SPLINE
SPL {X  -145.877, Y  +737.201, Z    +0.000, E1  +394.468, E3 -286395.030}
SPL {X  -152.550, Y  +719.721, Z    +0.000, E1  +387.728, E3 -286410.519}
SPL {X  -157.145, Y  +701.536, Z    +0.000, E1  +379.368, E3 -286419.974}
SPL {X  -159.035, Y  +688.952, Z    +0.000, E1  +372.676, E3 -286424.015}
SPL {X  -159.873, Y  +677.622, Z    +0.000, E1  +366.008, E3 -286426.087}
SPL {X  -159.990, Y  +671.638, Z    +0.000, E1  +361.925, E3 -286426.713}
SPL {X  -159.990, Y  +668.344, Z    +0.000, E1  +359.382, E3 -286426.906}
SPL {X  -159.990, Y  +664.070, Z    +0.000, E1  +354.975, E3 -286427.234}
SPL {X  -159.990, Y  +656.953, Z    +0.000, E1  +346.040, E3 -286428.300}
SPL {X  -159.990, Y  +644.589, Z    +0.000, E1  +330.989, E3 -286431.712}
SPL {X  -159.990, Y  +605.095, Z    +0.000, E1  +310.486, E3 -286456.803}
SPL {X  -159.990, Y  +546.155, Z    +0.000, E1  +305.539, E3 -286519.561}
SPL {X  -159.990, Y  +539.348, Z    +0.000, E1  +305.531, E3 -286529.865}
SPL {X  -159.990, Y  +530.752, Z    +0.000, E1  +305.518, E3 -286542.872}
SPL {X  -159.990, Y  +522.797, Z    +0.000, E1  +305.537, E3 -286554.956}
SPL {X  -159.990, Y  +515.332, Z    +0.000, E1  +305.526, E3 -286566.244}
SPL {X  -159.990, Y  +508.047, Z    +0.000, E1  +305.531, E3 -286577.261}
SPL {X  -159.990, Y  +499.403, Z    +0.000, E1  +305.488, E3 -286590.300}
SPL {X  -159.990, Y  +479.413, Z    +0.000, E1  +302.719, E3 -286601.446}
SPL {X  -159.990, Y  +454.926, Z    +0.000, E1  +299.433, E3 -286610.552}
SPL {X  -159.990, Y  +449.697, Z    +0.000, E1  +300.191, E3 -286622.015}
SPL {X  -159.990, Y  +444.026, Z    +0.000, E1  +301.072, E3 -286635.273}
SPL {X  -159.990, Y  +437.596, Z    +0.000, E1  +301.764, E3 -286648.015}
SPL {X  -159.990, Y  +432.883, Z    +0.000, E1  +302.386, E3 -286658.411}
SPL {X  -159.990, Y  +429.044, Z    +0.000, E1  +303.109, E3 -286668.302}
SPL {X  -159.990, Y  +425.222, Z    +0.000, E1  +304.101, E3 -286680.199}
SPL {X  -159.990, Y  +418.562, Z    +0.000, E1  +304.950, E3 -286695.356}
SPL {X  -159.990, Y  +410.722, Z    +0.000, E1  +305.100, E3 -286707.817}
SPL {X  -159.990, Y  +402.790, Z    +0.000, E1  +305.070, E3 -286719.592}
SPL {X  -159.990, Y  +391.119, Z    +0.000, E1  +305.052, E3 -286736.970}
SPL {X  -159.988, Y  +381.720, Z    +0.000, E1  +305.103, E3 -286751.077}
SPL {X  -159.786, Y  +374.425, Z    +0.000, E1  +305.121, E3 -286762.125}
SPL {X  -159.015, Y  +364.863, Z    +0.000, E1  +305.220, E3 -286777.142}
SPL {X  -157.966, Y  +357.131, Z    +0.000, E1  +305.441, E3 -286789.832}
SPL {X  -156.775, Y  +350.586, Z    +0.000, E1  +305.627, E3 -286800.806}
SPL {X  -155.397, Y  +344.442, Z    +0.000, E1  +305.886, E3 -286811.422}
SPL {X  -153.976, Y  +339.046, Z    +0.000, E1  +306.128, E3 -286820.914}
SPL {X  -152.417, Y  +333.859, Z    +0.000, E1  +306.416, E3 -286830.240}
SPL {X  -150.681, Y  +328.723, Z    +0.000, E1  +306.710, E3 -286839.616}
SPL {X  -148.661, Y  +323.366, Z    +0.000, E1  +307.100, E3 -286849.625}
SPL {X  -147.089, Y  +319.560, Z    +0.000, E1  +307.396, E3 -286856.840}
SPL {X  -145.161, Y  +315.232, Z    +0.000, E1  +307.745, E3 -286865.121}
SPL {X  -142.534, Y  +309.830, Z    +0.000, E1  +308.237, E3 -286875.626}
SPL {X  -132.342, Y  +292.599, Z    +0.000, E1  +315.826, E3 -286972.914}
ENDSPLINE

SPLINE
SPL {X  -151.238, Y  +330.309, Z    +0.000, E1  +330.693, E3 -287046.071}
SPL {X  -156.949, Y  +351.453, Z    +0.000, E1  +340.161, E3 -287058.231}
SPL {X  -159.024, Y  +364.945, Z    +0.000, E1  +347.297, E3 -287062.649}
SPL {X  -159.758, Y  +373.891, Z    +0.000, E1  +352.513, E3 -287064.538}
SPL {X  -159.985, Y  +381.208, Z    +0.000, E1  +357.184, E3 -287065.421}
SPL {X  -159.990, Y  +385.261, Z    +0.000, E1  +360.259, E3 -287065.691}
SPL {X  -159.990, Y  +388.094, Z    +0.000, E1  +363.012, E3 -287065.883}
SPL {X  -159.990, Y  +390.622, Z    +0.000, E1  +365.876, E3 -287066.122}
SPL {X  -159.990, Y  +394.493, Z    +0.000, E1  +370.512, E3 -287066.645}
SPL {X  -159.990, Y  +401.377, Z    +0.000, E1  +379.398, E3 -287068.099}
SPL {X  -159.990, Y  +411.365, Z    +0.000, E1  +390.630, E3 -287071.307}
SPL {X  -159.990, Y  +450.467, Z    +0.000, E1  +410.183, E3 -287094.956}
SPL {X  -159.990, Y  +509.934, Z    +0.000, E1  +414.923, E3 -287157.575}
SPL {X  -159.990, Y  +516.848, Z    +0.000, E1  +414.930, E3 -287167.863}
SPL {X  -159.990, Y  +524.818, Z    +0.000, E1  +414.933, E3 -287179.735}
SPL {X  -159.990, Y  +532.100, Z    +0.000, E1  +414.924, E3 -287190.588}
SPL {X  -159.990, Y  +539.391, Z    +0.000, E1  +414.933, E3 -287201.440}
SPL {X  -159.990, Y  +546.283, Z    +0.000, E1  +414.924, E3 -287211.712}
SPL {X  -159.990, Y  +553.734, Z    +0.000, E1  +414.938, E3 -287222.799}
SPL {X  -159.990, Y  +564.956, Z    +0.000, E1  +414.973, E3 -287239.470}
SPL {X  -159.990, Y  +577.902, Z    +0.000, E1  +414.969, E3 -287258.760}
SPL {X  -159.990, Y  +588.063, Z    +0.000, E1  +414.931, E3 -287273.951}
SPL {X  -159.990, Y  +595.273, Z    +0.000, E1  +414.928, E3 -287284.674}
SPL {X  -159.990, Y  +602.326, Z    +0.000, E1  +414.932, E3 -287295.174}
SPL {X  -159.990, Y  +609.708, Z    +0.000, E1  +414.930, E3 -287306.181}
SPL {X  -159.990, Y  +618.088, Z    +0.000, E1  +414.948, E3 -287318.610}
SPL {X  -159.990, Y  +625.928, Z    +0.000, E1  +414.931, E3 -287330.306}
SPL {X  -159.990, Y  +632.991, Z    +0.000, E1  +414.938, E3 -287340.809}
SPL {X  -159.990, Y  +639.033, Z    +0.000, E1  +414.931, E3 -287349.817}
SPL {X  -159.990, Y  +646.303, Z    +0.000, E1  +414.946, E3 -287360.604}
SPL {X  -159.990, Y  +656.335, Z    +0.000, E1  +414.969, E3 -287375.507}
SPL {X  -159.990, Y  +664.577, Z    +0.000, E1  +414.924, E3 -287387.884}
SPL {X  -159.989, Y  +672.128, Z    +0.000, E1  +414.946, E3 -287399.101}
SPL {X  -159.792, Y  +679.466, Z    +0.000, E1  +414.893, E3 -287410.259}
SPL {X  -159.330, Y  +686.016, Z    +0.000, E1  +414.837, E3 -287420.490}
SPL {X  -158.190, Y  +695.432, Z    +0.000, E1  +414.658, E3 -287435.686}
SPL {X  -157.027, Y  +702.151, Z    +0.000, E1  +414.415, E3 -287446.968}
SPL {X  -156.112, Y  +706.513, Z    +0.000, E1  +414.265, E3 -287454.402}
SPL {X  -154.917, Y  +711.470, Z    +0.000, E1  +414.052, E3 -287463.030}
SPL {X  -153.561, Y  +716.398, Z    +0.000, E1  +413.816, E3 -287471.751}
SPL {X  -151.715, Y  +722.287, Z    +0.000, E1  +413.503, E3 -287482.367}
SPL {X  -148.967, Y  +729.859, Z    +0.000, E1  +413.026, E3 -287496.359}
SPL {X  -145.862, Y  +737.236, Z    +0.000, E1  +412.427, E3 -287510.414}
SPL {X  -142.777, Y  +743.691, Z    +0.000, E1  +411.831, E3 -287522.957}
SPL {X  -132.301, Y  +761.463, Z    +0.000, E1  +405.510, E3 -287602.242}
ENDSPLINE

SPLINE
SPL {X  -145.877, Y  +737.201, Z    +0.000, E1  +394.468, E3 -287685.353}
SPL {X  -152.550, Y  +719.721, Z    +0.000, E1  +387.728, E3 -287700.842}
SPL {X  -157.145, Y  +701.536, Z    +0.000, E1  +379.368, E3 -287710.296}
SPL {X  -159.035, Y  +688.952, Z    +0.000, E1  +372.676, E3 -287714.337}
SPL {X  -159.756, Y  +680.154, Z    +0.000, E1  +367.520, E3 -287716.064}
SPL {X  -159.986, Y  +672.560, Z    +0.000, E1  +362.636, E3 -287716.962}
SPL {X  -159.990, Y  +668.344, Z    +0.000, E1  +359.382, E3 -287717.228}
SPL {X  -159.990, Y  +664.070, Z    +0.000, E1  +354.975, E3 -287717.556}
SPL {X  -159.990, Y  +656.953, Z    +0.000, E1  +346.040, E3 -287718.623}
SPL {X  -159.990, Y  +644.589, Z    +0.000, E1  +330.989, E3 -287722.034}
SPL {X  -159.990, Y  +605.095, Z    +0.000, E1  +310.486, E3 -287747.125}
SPL {X  -159.990, Y  +546.155, Z    +0.000, E1  +305.539, E3 -287809.884}
SPL {X  -159.990, Y  +539.348, Z    +0.000, E1  +305.531, E3 -287820.188}
SPL {X  -159.990, Y  +530.752, Z    +0.000, E1  +305.518, E3 -287833.195}
SPL {X  -159.990, Y  +522.797, Z    +0.000, E1  +305.537, E3 -287845.278}
SPL {X  -159.990, Y  +515.332, Z    +0.000, E1  +305.526, E3 -287856.567}
SPL {X  -159.990, Y  +508.047, Z    +0.000, E1  +305.531, E3 -287867.584}
SPL {X  -159.990, Y  +499.403, Z    +0.000, E1  +305.488, E3 -287880.623}
SPL {X  -159.990, Y  +479.413, Z    +0.000, E1  +302.719, E3 -287891.768}
SPL {X  -159.990, Y  +454.926, Z    +0.000, E1  +299.433, E3 -287900.875}
SPL {X  -159.990, Y  +449.697, Z    +0.000, E1  +300.191, E3 -287912.337}
SPL {X  -159.990, Y  +445.847, Z    +0.000, E1  +300.905, E3 -287921.960}
SPL {X  -159.990, Y  +439.266, Z    +0.000, E1  +301.568, E3 -287935.044}
SPL {X  -159.990, Y  +432.883, Z    +0.000, E1  +302.386, E3 -287948.734}
SPL {X  -159.990, Y  +429.044, Z    +0.000, E1  +303.109, E3 -287958.624}
SPL {X  -159.990, Y  +425.222, Z    +0.000, E1  +304.101, E3 -287970.521}
SPL {X  -159.990, Y  +420.083, Z    +0.000, E1  +304.918, E3 -287983.097}
SPL {X  -159.990, Y  +412.567, Z    +0.000, E1  +305.072, E3 -287995.321}
SPL {X  -159.990, Y  +402.790, Z    +0.000, E1  +305.070, E3 -288009.915}
SPL {X  -159.990, Y  +391.119, Z    +0.000, E1  +305.052, E3 -288027.293}
SPL {X  -159.988, Y  +381.720, Z    +0.000, E1  +305.103, E3 -288041.400}
SPL {X  -159.786, Y  +374.425, Z    +0.000, E1  +305.121, E3 -288052.448}
SPL {X  -159.015, Y  +364.863, Z    +0.000, E1  +305.220, E3 -288067.464}
SPL {X  -157.966, Y  +357.131, Z    +0.000, E1  +305.441, E3 -288080.155}
SPL {X  -156.775, Y  +350.586, Z    +0.000, E1  +305.627, E3 -288091.129}
SPL {X  -155.027, Y  +342.959, Z    +0.000, E1  +305.926, E3 -288104.302}
SPL {X  -152.882, Y  +335.340, Z    +0.000, E1  +306.305, E3 -288117.844}
SPL {X  -150.681, Y  +328.723, Z    +0.000, E1  +306.710, E3 -288129.939}
SPL {X  -148.661, Y  +323.366, Z    +0.000, E1  +307.100, E3 -288139.948}
SPL {X  -147.089, Y  +319.560, Z    +0.000, E1  +307.396, E3 -288147.163}
SPL {X  -145.161, Y  +315.232, Z    +0.000, E1  +307.745, E3 -288155.443}
SPL {X  -142.534, Y  +309.830, Z    +0.000, E1  +308.237, E3 -288165.948}
SPL {X  -132.342, Y  +292.599, Z    +0.000, E1  +315.826, E3 -288263.237}
ENDSPLINE

SPLINE
SPL {X  -151.238, Y  +330.309, Z    +0.000, E1  +330.693, E3 -288336.393}
SPL {X  -156.949, Y  +351.453, Z    +0.000, E1  +340.161, E3 -288348.554}
SPL {X  -159.024, Y  +364.945, Z    +0.000, E1  +347.297, E3 -288352.972}
SPL {X  -159.878, Y  +376.512, Z    +0.000, E1  +354.071, E3 -288355.223}
SPL {X  -159.990, Y  +383.659, Z    +0.000, E1  +358.950, E3 -288355.918}
SPL {X  -159.990, Y  +387.327, Z    +0.000, E1  +362.137, E3 -288356.151}
SPL {X  -159.990, Y  +390.622, Z    +0.000, E1  +365.876, E3 -288356.444}
SPL {X  -159.990, Y  +394.493, Z    +0.000, E1  +370.512, E3 -288356.967}
SPL {X  -159.990, Y  +401.377, Z    +0.000, E1  +379.398, E3 -288358.422}
SPL {X  -159.990, Y  +411.365, Z    +0.000, E1  +390.630, E3 -288361.630}
SPL {X  -159.990, Y  +450.467, Z    +0.000, E1  +410.183, E3 -288385.279}
SPL {X  -159.990, Y  +509.934, Z    +0.000, E1  +414.923, E3 -288447.898}
SPL {X  -159.990, Y  +516.848, Z    +0.000, E1  +414.930, E3 -288458.186}
SPL {X  -159.990, Y  +524.818, Z    +0.000, E1  +414.933, E3 -288470.058}
SPL {X  -159.990, Y  +532.100, Z    +0.000, E1  +414.924, E3 -288480.911}
SPL {X  -159.990, Y  +539.391, Z    +0.000, E1  +414.933, E3 -288491.763}
SPL {X  -159.990, Y  +546.283, Z    +0.000, E1  +414.924, E3 -288502.034}
SPL {X  -159.990, Y  +553.734, Z    +0.000, E1  +414.938, E3 -288513.121}
SPL {X  -159.990, Y  +564.956, Z    +0.000, E1  +414.973, E3 -288529.792}
SPL {X  -159.990, Y  +577.902, Z    +0.000, E1  +414.969, E3 -288549.082}
SPL {X  -159.990, Y  +588.063, Z    +0.000, E1  +414.931, E3 -288564.273}
SPL {X  -159.990, Y  +595.273, Z    +0.000, E1  +414.928, E3 -288574.997}
SPL {X  -159.990, Y  +602.326, Z    +0.000, E1  +414.932, E3 -288585.497}
SPL {X  -159.990, Y  +609.708, Z    +0.000, E1  +414.930, E3 -288596.504}
SPL {X  -159.990, Y  +618.088, Z    +0.000, E1  +414.948, E3 -288608.933}
SPL {X  -159.990, Y  +625.928, Z    +0.000, E1  +414.931, E3 -288620.629}
SPL {X  -159.990, Y  +635.803, Z    +0.000, E1  +414.980, E3 -288635.257}
SPL {X  -159.990, Y  +646.303, Z    +0.000, E1  +414.946, E3 -288650.927}
SPL {X  -159.990, Y  +653.312, Z    +0.000, E1  +414.932, E3 -288661.379}
SPL {X  -159.990, Y  +658.943, Z    +0.000, E1  +414.931, E3 -288669.777}
SPL {X  -159.990, Y  +667.151, Z    +0.000, E1  +414.954, E3 -288681.995}
SPL {X  -159.885, Y  +677.285, Z    +0.000, E1  +414.936, E3 -288697.191}
SPL {X  -159.482, Y  +684.244, Z    +0.000, E1  +414.840, E3 -288708.043}
SPL {X  -158.805, Y  +690.934, Z    +0.000, E1  +414.742, E3 -288718.692}
SPL {X  -157.890, Y  +697.337, Z    +0.000, E1  +414.571, E3 -288729.214}
SPL {X  -156.492, Y  +704.774, Z    +0.000, E1  +414.365, E3 -288741.692}
SPL {X  -154.917, Y  +711.470, Z    +0.000, E1  +414.052, E3 -288753.352}
SPL {X  -153.561, Y  +716.398, Z    +0.000, E1  +413.816, E3 -288762.074}
SPL {X  -151.715, Y  +722.287, Z    +0.000, E1  +413.503, E3 -288772.690}
SPL {X  -148.967, Y  +729.859, Z    +0.000, E1  +413.026, E3 -288786.682}
SPL {X  -145.862, Y  +737.236, Z    +0.000, E1  +412.427, E3 -288800.736}
SPL {X  -142.777, Y  +743.691, Z    +0.000, E1  +411.831, E3 -288813.279}
SPL {X  -132.301, Y  +761.463, Z    +0.000, E1  +405.510, E3 -288892.564}
ENDSPLINE

SPLINE
SPL {X  -145.877, Y  +737.201, Z    +0.000, E1  +394.468, E3 -288975.675}
SPL {X  -152.550, Y  +719.721, Z    +0.000, E1  +387.728, E3 -288991.164}
SPL {X  -157.145, Y  +701.536, Z    +0.000, E1  +379.368, E3 -289000.619}
SPL {X  -159.035, Y  +688.952, Z    +0.000, E1  +372.676, E3 -289004.660}
SPL {X  -159.756, Y  +680.154, Z    +0.000, E1  +367.520, E3 -289006.386}
SPL {X  -159.986, Y  +672.560, Z    +0.000, E1  +362.636, E3 -289007.284}
SPL {X  -159.990, Y  +668.344, Z    +0.000, E1  +359.382, E3 -289007.551}
SPL {X  -159.990, Y  +664.070, Z    +0.000, E1  +354.975, E3 -289007.879}
SPL {X  -159.990, Y  +656.953, Z    +0.000, E1  +346.040, E3 -289008.946}
SPL {X  -159.990, Y  +644.589, Z    +0.000, E1  +330.989, E3 -289012.357}
SPL {X  -159.990, Y  +605.095, Z    +0.000, E1  +310.486, E3 -289037.448}
SPL {X  -159.990, Y  +546.155, Z    +0.000, E1  +305.539, E3 -289100.206}
SPL {X  -159.990, Y  +539.348, Z    +0.000, E1  +305.531, E3 -289110.510}
SPL {X  -159.990, Y  +530.752, Z    +0.000, E1  +305.518, E3 -289123.518}
SPL {X  -159.990, Y  +522.797, Z    +0.000, E1  +305.537, E3 -289135.601}
SPL {X  -159.990, Y  +515.332, Z    +0.000, E1  +305.526, E3 -289146.890}
SPL {X  -159.990, Y  +508.047, Z    +0.000, E1  +305.531, E3 -289157.906}
SPL {X  -159.990, Y  +501.296, Z    +0.000, E1  +305.518, E3 -289168.128}
SPL {X  -159.990, Y  +487.558, Z    +0.000, E1  +304.151, E3 -289179.758}
SPL {X  -159.990, Y  +454.926, Z    +0.000, E1  +299.433, E3 -289191.197}
SPL {X  -159.990, Y  +449.697, Z    +0.000, E1  +300.191, E3 -289202.660}
SPL {X  -159.990, Y  +445.847, Z    +0.000, E1  +300.905, E3 -289212.283}
SPL {X  -159.990, Y  +439.266, Z    +0.000, E1  +301.568, E3 -289225.366}
SPL {X  -159.990, Y  +432.883, Z    +0.000, E1  +302.386, E3 -289239.057}
SPL {X  -159.990, Y  +429.044, Z    +0.000, E1  +303.109, E3 -289248.947}
SPL {X  -159.990, Y  +425.222, Z    +0.000, E1  +304.101, E3 -289260.844}
SPL {X  -159.990, Y  +418.562, Z    +0.000, E1  +304.950, E3 -289276.002}
SPL {X  -159.990, Y  +407.911, Z    +0.000, E1  +305.062, E3 -289292.593}
SPL {X  -159.990, Y  +400.284, Z    +0.000, E1  +305.103, E3 -289304.027}
SPL {X  -159.990, Y  +391.119, Z    +0.000, E1  +305.052, E3 -289317.615}
SPL {X  -159.988, Y  +381.720, Z    +0.000, E1  +305.103, E3 -289331.722}
SPL {X  -159.786, Y  +374.425, Z    +0.000, E1  +305.121, E3 -289342.771}
SPL {X  -159.015, Y  +364.863, Z    +0.000, E1  +305.220, E3 -289357.787}
SPL {X  -157.966, Y  +357.131, Z    +0.000, E1  +305.441, E3 -289370.477}
SPL {X  -156.775, Y  +350.586, Z    +0.000, E1  +305.627, E3 -289381.451}
SPL {X  -155.027, Y  +342.959, Z    +0.000, E1  +305.926, E3 -289394.624}
SPL {X  -152.882, Y  +335.340, Z    +0.000, E1  +306.305, E3 -289408.167}
SPL {X  -150.681, Y  +328.723, Z    +0.000, E1  +306.710, E3 -289420.261}
SPL {X  -148.661, Y  +323.366, Z    +0.000, E1  +307.100, E3 -289430.270}
SPL {X  -147.089, Y  +319.560, Z    +0.000, E1  +307.396, E3 -289437.485}
SPL {X  -145.161, Y  +315.232, Z    +0.000, E1  +307.745, E3 -289445.766}
SPL {X  -142.534, Y  +309.830, Z    +0.000, E1  +308.237, E3 -289456.271}
SPL {X  -132.342, Y  +292.599, Z    +0.000, E1  +315.826, E3 -289553.559}
ENDSPLINE

SPLINE
SPL {X  -151.238, Y  +330.309, Z    +0.000, E1  +330.693, E3 -289626.716}
SPL {X  -156.949, Y  +351.453, Z    +0.000, E1  +340.161, E3 -289638.877}
SPL {X  -159.024, Y  +364.945, Z    +0.000, E1  +347.297, E3 -289643.294}
SPL {X  -159.758, Y  +373.891, Z    +0.000, E1  +352.513, E3 -289645.183}
SPL {X  -159.985, Y  +381.208, Z    +0.000, E1  +357.184, E3 -289646.066}
SPL {X  -159.990, Y  +384.493, Z    +0.000, E1  +359.676, E3 -289646.291}
SPL {X  -159.990, Y  +387.327, Z    +0.000, E1  +362.137, E3 -289646.473}
SPL {X  -159.990, Y  +392.053, Z    +0.000, E1  +367.477, E3 -289646.938}
SPL {X  -159.990, Y  +396.158, Z    +0.000, E1  +372.775, E3 -289647.564}
SPL {X  -159.990, Y  +401.377, Z    +0.000, E1  +379.398, E3 -289648.744}
SPL {X  -159.990, Y  +411.365, Z    +0.000, E1  +390.630, E3 -289651.953}
SPL {X  -159.990, Y  +450.467, Z    +0.000, E1  +410.183, E3 -289675.602}
SPL {X  -159.990, Y  +509.934, Z    +0.000, E1  +414.923, E3 -289738.220}
SPL {X  -159.990, Y  +516.848, Z    +0.000, E1  +414.930, E3 -289748.508}
SPL {X  -159.990, Y  +524.818, Z    +0.000, E1  +414.933, E3 -289760.380}
SPL {X  -159.990, Y  +532.100, Z    +0.000, E1  +414.924, E3 -289771.233}
SPL {X  -159.990, Y  +539.391, Z    +0.000, E1  +414.933, E3 -289782.085}
SPL {X  -159.990, Y  +546.283, Z    +0.000, E1  +414.924, E3 -289792.357}
SPL {X  -159.990, Y  +553.734, Z    +0.000, E1  +414.938, E3 -289803.444}
SPL {X  -159.990, Y  +564.956, Z    +0.000, E1  +414.973, E3 -289820.115}
SPL {X  -159.990, Y  +577.902, Z    +0.000, E1  +414.969, E3 -289839.405}
SPL {X  -159.990, Y  +588.063, Z    +0.000, E1  +414.931, E3 -289854.596}
SPL {X  -159.990, Y  +595.273, Z    +0.000, E1  +414.928, E3 -289865.319}
SPL {X  -159.990, Y  +602.326, Z    +0.000, E1  +414.932, E3 -289875.820}
SPL {X  -159.990, Y  +609.708, Z    +0.000, E1  +414.930, E3 -289886.826}
SPL {X  -159.990, Y  +618.088, Z    +0.000, E1  +414.948, E3 -289899.255}
SPL {X  -159.990, Y  +625.928, Z    +0.000, E1  +414.931, E3 -289910.951}
SPL {X  -159.990, Y  +635.803, Z    +0.000, E1  +414.980, E3 -289925.579}
SPL {X  -159.990, Y  +646.303, Z    +0.000, E1  +414.946, E3 -289941.250}
SPL {X  -159.990, Y  +656.335, Z    +0.000, E1  +414.969, E3 -289956.152}
SPL {X  -159.990, Y  +664.577, Z    +0.000, E1  +414.924, E3 -289968.529}
SPL {X  -159.989, Y  +672.128, Z    +0.000, E1  +414.946, E3 -289979.746}
SPL {X  -159.636, Y  +682.136, Z    +0.000, E1  +414.901, E3 -289995.004}
SPL {X  -158.805, Y  +690.934, Z    +0.000, E1  +414.742, E3 -290009.015}
SPL {X  -157.890, Y  +697.337, Z    +0.000, E1  +414.571, E3 -290019.536}
SPL {X  -156.492, Y  +704.774, Z    +0.000, E1  +414.365, E3 -290032.015}
SPL {X  -154.917, Y  +711.470, Z    +0.000, E1  +414.052, E3 -290043.675}
SPL {X  -153.204, Y  +717.603, Z    +0.000, E1  +413.775, E3 -290054.521}
SPL {X  -151.355, Y  +723.351, Z    +0.000, E1  +413.415, E3 -290064.992}
SPL {X  -148.967, Y  +729.859, Z    +0.000, E1  +413.026, E3 -290077.004}
SPL {X  -145.862, Y  +737.236, Z    +0.000, E1  +412.427, E3 -290091.059}
SPL {X  -142.777, Y  +743.691, Z    +0.000, E1  +411.831, E3 -290103.602}
SPL {X  -132.301, Y  +761.463, Z    +0.000, E1  +405.510, E3 -290182.887}
ENDSPLINE

SPLINE
SPL {X  -145.877, Y  +737.201, Z    +0.000, E1  +394.468, E3 -290265.998}
SPL {X  -152.550, Y  +719.721, Z    +0.000, E1  +387.728, E3 -290281.487}
SPL {X  -157.145, Y  +701.536, Z    +0.000, E1  +379.368, E3 -290290.942}
SPL {X  -159.035, Y  +688.952, Z    +0.000, E1  +372.676, E3 -290294.983}
SPL {X  -159.756, Y  +680.154, Z    +0.000, E1  +367.520, E3 -290296.709}
SPL {X  -159.986, Y  +672.560, Z    +0.000, E1  +362.636, E3 -290297.607}
SPL {X  -159.990, Y  +669.364, Z    +0.000, E1  +360.170, E3 -290297.815}
SPL {X  -159.990, Y  +667.647, Z    +0.000, E1  +358.660, E3 -290297.913}
SPL {X  -159.990, Y  +664.070, Z    +0.000, E1  +354.975, E3 -290298.202}
SPL {X  -159.990, Y  +656.953, Z    +0.000, E1  +346.040, E3 -290299.268}
SPL {X  -159.990, Y  +644.589, Z    +0.000, E1  +330.989, E3 -290302.680}
SPL {X  -159.990, Y  +605.095, Z    +0.000, E1  +310.486, E3 -290327.771}
SPL {X  -159.990, Y  +546.155, Z    +0.000, E1  +305.539, E3 -290390.529}
SPL {X  -159.990, Y  +539.348, Z    +0.000, E1  +305.531, E3 -290400.833}
SPL {X  -159.990, Y  +530.752, Z    +0.000, E1  +305.518, E3 -290413.840}
SPL {X  -159.990, Y  +522.797, Z    +0.000, E1  +305.537, E3 -290425.923}
SPL {X  -159.990, Y  +515.332, Z    +0.000, E1  +305.526, E3 -290437.212}
SPL {X  -159.990, Y  +508.047, Z    +0.000, E1  +305.531, E3 -290448.229}
SPL {X  -159.990, Y  +499.403, Z    +0.000, E1  +305.488, E3 -290461.268}
SPL {X  -159.990, Y  +479.413, Z    +0.000, E1  +302.719, E3 -290472.413}
SPL {X  -159.990, Y  +454.926, Z    +0.000, E1  +299.433, E3 -290481.520}
SPL {X  -159.990, Y  +449.697, Z    +0.000, E1  +300.191, E3 -290492.982}
SPL {X  -159.990, Y  +445.847, Z    +0.000, E1  +300.905, E3 -290502.605}
SPL {X  -159.990, Y  +439.266, Z    +0.000, E1  +301.568, E3 -290515.689}
SPL {X  -159.990, Y  +432.883, Z    +0.000, E1  +302.386, E3 -290529.379}
SPL {X  -159.990, Y  +429.044, Z    +0.000, E1  +303.109, E3 -290539.269}
SPL {X  -159.990, Y  +425.222, Z    +0.000, E1  +304.101, E3 -290551.166}
SPL {X  -159.990, Y  +420.083, Z    +0.000, E1  +304.918, E3 -290563.742}
SPL {X  -159.990, Y  +412.567, Z    +0.000, E1  +305.072, E3 -290575.966}
SPL {X  -159.990, Y  +402.790, Z    +0.000, E1  +305.070, E3 -290590.560}
SPL {X  -159.990, Y  +391.119, Z    +0.000, E1  +305.052, E3 -290607.938}
SPL {X  -159.988, Y  +381.720, Z    +0.000, E1  +305.103, E3 -290622.045}
SPL {X  -159.786, Y  +374.425, Z    +0.000, E1  +305.121, E3 -290633.093}
SPL {X  -159.015, Y  +364.863, Z    +0.000, E1  +305.220, E3 -290648.109}
SPL {X  -157.966, Y  +357.131, Z    +0.000, E1  +305.441, E3 -290660.800}
SPL {X  -156.775, Y  +350.586, Z    +0.000, E1  +305.627, E3 -290671.774}
SPL {X  -155.027, Y  +342.959, Z    +0.000, E1  +305.926, E3 -290684.947}
SPL {X  -152.882, Y  +335.340, Z    +0.000, E1  +306.305, E3 -290698.489}
SPL {X  -150.681, Y  +328.723, Z    +0.000, E1  +306.710, E3 -290710.584}
SPL {X  -148.661, Y  +323.366, Z    +0.000, E1  +307.100, E3 -290720.593}
SPL {X  -147.089, Y  +319.560, Z    +0.000, E1  +307.396, E3 -290727.808}
SPL {X  -145.161, Y  +315.232, Z    +0.000, E1  +307.745, E3 -290736.088}
SPL {X  -142.534, Y  +309.830, Z    +0.000, E1  +308.237, E3 -290746.594}
SPL {X  -132.342, Y  +292.599, Z    +0.000, E1  +315.826, E3 -290843.882}
ENDSPLINE

SPLINE
SPL {X  -151.238, Y  +330.309, Z    +0.000, E1  +330.693, E3 -290917.038}
SPL {X  -156.949, Y  +351.453, Z    +0.000, E1  +340.161, E3 -290929.199}
SPL {X  -159.024, Y  +364.945, Z    +0.000, E1  +347.297, E3 -290933.617}
SPL {X  -159.878, Y  +376.512, Z    +0.000, E1  +354.071, E3 -290935.869}
SPL {X  -159.990, Y  +383.659, Z    +0.000, E1  +358.950, E3 -290936.563}
SPL {X  -159.990, Y  +387.327, Z    +0.000, E1  +362.137, E3 -290936.796}
SPL {X  -159.990, Y  +390.622, Z    +0.000, E1  +365.876, E3 -290937.089}
SPL {X  -159.990, Y  +394.493, Z    +0.000, E1  +370.512, E3 -290937.612}
SPL {X  -159.990, Y  +401.377, Z    +0.000, E1  +379.398, E3 -290939.067}
SPL {X  -159.990, Y  +411.365, Z    +0.000, E1  +390.630, E3 -290942.275}
SPL {X  -159.990, Y  +450.467, Z    +0.000, E1  +410.183, E3 -290965.924}
SPL {X  -159.990, Y  +509.934, Z    +0.000, E1  +414.923, E3 -291028.543}
SPL {X  -159.990, Y  +516.848, Z    +0.000, E1  +414.930, E3 -291038.831}
SPL {X  -159.990, Y  +524.818, Z    +0.000, E1  +414.933, E3 -291050.703}
SPL {X  -159.990, Y  +532.100, Z    +0.000, E1  +414.924, E3 -291061.556}
SPL {X  -159.990, Y  +539.391, Z    +0.000, E1  +414.933, E3 -291072.408}
SPL {X  -159.990, Y  +546.283, Z    +0.000, E1  +414.924, E3 -291082.680}
SPL {X  -159.990, Y  +553.734, Z    +0.000, E1  +414.938, E3 -291093.766}
SPL {X  -159.990, Y  +560.657, Z    +0.000, E1  +414.914, E3 -291104.127}
SPL {X  -159.990, Y  +567.311, Z    +0.000, E1  +414.931, E3 -291114.012}
SPL {X  -159.990, Y  +577.902, Z    +0.000, E1  +414.969, E3 -291129.727}
SPL {X  -159.990, Y  +588.063, Z    +0.000, E1  +414.931, E3 -291144.918}
SPL {X  -159.990, Y  +595.273, Z    +0.000, E1  +414.928, E3 -291155.642}
SPL {X  -159.990, Y  +602.326, Z    +0.000, E1  +414.932, E3 -291166.142}
SPL {X  -159.990, Y  +609.708, Z    +0.000, E1  +414.930, E3 -291177.149}
SPL {X  -159.990, Y  +616.306, Z    +0.000, E1  +414.927, E3 -291186.962}
SPL {X  -159.990, Y  +624.320, Z    +0.000, E1  +414.952, E3 -291198.845}
SPL {X  -159.990, Y  +632.991, Z    +0.000, E1  +414.938, E3 -291211.777}
SPL {X  -159.990, Y  +639.033, Z    +0.000, E1  +414.931, E3 -291220.784}
SPL {X  -159.990, Y  +646.303, Z    +0.000, E1  +414.946, E3 -291231.572}
SPL {X  -159.990, Y  +656.335, Z    +0.000, E1  +414.969, E3 -291246.474}
SPL {X  -159.990, Y  +664.577, Z    +0.000, E1  +414.924, E3 -291258.852}
SPL {X  -159.989, Y  +672.128, Z    +0.000, E1  +414.946, E3 -291270.068}
SPL {X  -159.792, Y  +679.466, Z    +0.000, E1  +414.893, E3 -291281.226}
SPL {X  -159.330, Y  +686.016, Z    +0.000, E1  +414.837, E3 -291291.457}
SPL {X  -158.190, Y  +695.432, Z    +0.000, E1  +414.658, E3 -291306.654}
SPL {X  -157.027, Y  +702.151, Z    +0.000, E1  +414.415, E3 -291317.936}
SPL {X  -156.112, Y  +706.513, Z    +0.000, E1  +414.265, E3 -291325.370}
SPL {X  -154.917, Y  +711.470, Z    +0.000, E1  +414.052, E3 -291333.997}
SPL {X  -153.561, Y  +716.398, Z    +0.000, E1  +413.816, E3 -291342.719}
SPL {X  -151.715, Y  +722.287, Z    +0.000, E1  +413.503, E3 -291353.335}
SPL {X  -149.700, Y  +727.952, Z    +0.000, E1  +413.118, E3 -291363.809}
SPL {X  -147.376, Y  +733.767, Z    +0.000, E1  +412.706, E3 -291374.759}
SPL {X  -145.109, Y  +738.881, Z    +0.000, E1  +412.243, E3 -291384.606}
SPL {X  -142.777, Y  +743.691, Z    +0.000, E1  +411.831, E3 -291393.925}
SPL {X  -132.301, Y  +761.463, Z    +0.000, E1  +405.510, E3 -291473.209}
ENDSPLINE

SPLINE
SPL {X  -145.877, Y  +737.201, Z    +0.000, E1  +394.468, E3 -291556.320}
SPL {X  -152.550, Y  +719.721, Z    +0.000, E1  +387.728, E3 -291571.810}
SPL {X  -157.145, Y  +701.536, Z    +0.000, E1  +379.368, E3 -291581.264}
SPL {X  -159.035, Y  +688.952, Z    +0.000, E1  +372.676, E3 -291585.305}
SPL {X  -159.873, Y  +677.622, Z    +0.000, E1  +366.008, E3 -291587.377}
SPL {X  -159.990, Y  +671.638, Z    +0.000, E1  +361.925, E3 -291588.004}
SPL {X  -159.990, Y  +668.344, Z    +0.000, E1  +359.382, E3 -291588.196}
SPL {X  -159.990, Y  +664.070, Z    +0.000, E1  +354.975, E3 -291588.524}
SPL {X  -159.990, Y  +658.737, Z    +0.000, E1  +348.199, E3 -291589.230}
SPL {X  -159.990, Y  +652.023, Z    +0.000, E1  +339.551, E3 -291590.715}
SPL {X  -159.990, Y  +641.935, Z    +0.000, E1  +328.152, E3 -291593.887}
SPL {X  -159.990, Y  +605.095, Z    +0.000, E1  +310.486, E3 -291618.093}
SPL {X  -159.990, Y  +546.155, Z    +0.000, E1  +305.539, E3 -291680.852}
SPL {X  -159.990, Y  +539.348, Z    +0.000, E1  +305.531, E3 -291691.155}
SPL {X  -159.990, Y  +530.752, Z    +0.000, E1  +305.518, E3 -291704.163}
SPL {X  -159.990, Y  +522.797, Z    +0.000, E1  +305.537, E3 -291716.246}
SPL {X  -159.990, Y  +515.332, Z    +0.000, E1  +305.526, E3 -291727.535}
SPL {X  -159.990, Y  +508.047, Z    +0.000, E1  +305.531, E3 -291738.552}
SPL {X  -159.990, Y  +501.296, Z    +0.000, E1  +305.518, E3 -291748.773}
SPL {X  -159.990, Y  +487.558, Z    +0.000, E1  +304.151, E3 -291760.403}
SPL {X  -159.990, Y  +454.926, Z    +0.000, E1  +299.433, E3 -291771.843}
SPL {X  -159.990, Y  +449.697, Z    +0.000, E1  +300.191, E3 -291783.305}
SPL {X  -159.990, Y  +445.847, Z    +0.000, E1  +300.905, E3 -291792.928}
SPL {X  -159.990, Y  +439.266, Z    +0.000, E1  +301.568, E3 -291806.011}
SPL {X  -159.990, Y  +432.883, Z    +0.000, E1  +302.386, E3 -291819.702}
SPL {X  -159.990, Y  +429.044, Z    +0.000, E1  +303.109, E3 -291829.592}
SPL {X  -159.990, Y  +425.222, Z    +0.000, E1  +304.101, E3 -291841.489}
SPL {X  -159.990, Y  +418.562, Z    +0.000, E1  +304.950, E3 -291856.647}
SPL {X  -159.990, Y  +407.911, Z    +0.000, E1  +305.062, E3 -291873.238}
SPL {X  -159.990, Y  +400.284, Z    +0.000, E1  +305.103, E3 -291884.672}
SPL {X  -159.990, Y  +391.119, Z    +0.000, E1  +305.052, E3 -291898.260}
SPL {X  -159.988, Y  +381.720, Z    +0.000, E1  +305.103, E3 -291912.368}
SPL {X  -159.786, Y  +374.425, Z    +0.000, E1  +305.121, E3 -291923.416}
SPL {X  -159.015, Y  +364.863, Z    +0.000, E1  +305.220, E3 -291938.432}
SPL {X  -157.966, Y  +357.131, Z    +0.000, E1  +305.441, E3 -291951.122}
SPL {X  -156.775, Y  +350.586, Z    +0.000, E1  +305.627, E3 -291962.096}
SPL {X  -155.027, Y  +342.959, Z    +0.000, E1  +305.926, E3 -291975.269}
SPL {X  -152.882, Y  +335.340, Z    +0.000, E1  +306.305, E3 -291988.812}
SPL {X  -150.681, Y  +328.723, Z    +0.000, E1  +306.710, E3 -292000.906}
SPL {X  -148.661, Y  +323.366, Z    +0.000, E1  +307.100, E3 -292010.916}
SPL {X  -147.089, Y  +319.560, Z    +0.000, E1  +307.396, E3 -292018.131}
SPL {X  -145.161, Y  +315.232, Z    +0.000, E1  +307.745, E3 -292026.411}
SPL {X  -142.534, Y  +309.830, Z    +0.000, E1  +308.237, E3 -292036.916}
SPL {X  -132.342, Y  +292.599, Z    +0.000, E1  +315.826, E3 -292134.204}
ENDSPLINE

SPLINE
SPL {X  -151.238, Y  +330.309, Z    +0.000, E1  +330.693, E3 -292207.361}
SPL {X  -156.949, Y  +351.453, Z    +0.000, E1  +340.161, E3 -292219.522}
SPL {X  -159.024, Y  +364.945, Z    +0.000, E1  +347.297, E3 -292223.940}
SPL {X  -159.878, Y  +376.512, Z    +0.000, E1  +354.071, E3 -292226.191}
SPL {X  -159.990, Y  +383.659, Z    +0.000, E1  +358.950, E3 -292226.886}
SPL {X  -159.990, Y  +387.327, Z    +0.000, E1  +362.137, E3 -292227.119}
SPL {X  -159.990, Y  +390.622, Z    +0.000, E1  +365.876, E3 -292227.412}
SPL {X  -159.990, Y  +394.493, Z    +0.000, E1  +370.512, E3 -292227.935}
SPL {X  -159.990, Y  +401.377, Z    +0.000, E1  +379.398, E3 -292229.389}
SPL {X  -159.990, Y  +411.365, Z    +0.000, E1  +390.630, E3 -292232.598}
SPL {X  -159.990, Y  +450.467, Z    +0.000, E1  +410.183, E3 -292256.247}
SPL {X  -159.990, Y  +509.934, Z    +0.000, E1  +414.923, E3 -292318.866}
SPL {X  -159.990, Y  +516.848, Z    +0.000, E1  +414.930, E3 -292329.154}
SPL {X  -159.990, Y  +524.818, Z    +0.000, E1  +414.933, E3 -292341.025}
SPL {X  -159.990, Y  +532.100, Z    +0.000, E1  +414.924, E3 -292351.879}
SPL {X  -159.990, Y  +539.391, Z    +0.000, E1  +414.933, E3 -292362.731}
SPL {X  -159.990, Y  +546.283, Z    +0.000, E1  +414.924, E3 -292373.002}
SPL {X  -159.990, Y  +553.734, Z    +0.000, E1  +414.938, E3 -292384.089}
SPL {X  -159.990, Y  +560.657, Z    +0.000, E1  +414.914, E3 -292394.450}
SPL {X  -159.990, Y  +567.311, Z    +0.000, E1  +414.931, E3 -292404.334}
SPL {X  -159.990, Y  +575.140, Z    +0.000, E1  +414.928, E3 -292415.994}
SPL {X  -159.990, Y  +581.046, Z    +0.000, E1  +414.920, E3 -292424.806}
SPL {X  -159.990, Y  +588.063, Z    +0.000, E1  +414.931, E3 -292435.241}
SPL {X  -159.990, Y  +595.273, Z    +0.000, E1  +414.928, E3 -292445.964}
SPL {X  -159.990, Y  +602.326, Z    +0.000, E1  +414.932, E3 -292456.465}
SPL {X  -159.990, Y  +609.708, Z    +0.000, E1  +414.930, E3 -292467.471}
SPL {X  -159.990, Y  +618.088, Z    +0.000, E1  +414.948, E3 -292479.900}
SPL {X  -159.990, Y  +625.928, Z    +0.000, E1  +414.931, E3 -292491.596}
SPL {X  -159.990, Y  +632.991, Z    +0.000, E1  +414.938, E3 -292502.099}
SPL {X  -159.990, Y  +639.033, Z    +0.000, E1  +414.931, E3 -292511.107}
SPL {X  -159.990, Y  +646.303, Z    +0.000, E1  +414.946, E3 -292521.895}
SPL {X  -159.990, Y  +656.335, Z    +0.000, E1  +414.969, E3 -292536.797}
SPL {X  -159.990, Y  +664.577, Z    +0.000, E1  +414.924, E3 -292549.174}
SPL {X  -159.989, Y  +672.128, Z    +0.000, E1  +414.946, E3 -292560.391}
SPL {X  -159.636, Y  +682.136, Z    +0.000, E1  +414.901, E3 -292575.649}
SPL {X  -158.805, Y  +690.934, Z    +0.000, E1  +414.742, E3 -292589.660}
SPL {X  -157.890, Y  +697.337, Z    +0.000, E1  +414.571, E3 -292600.181}
SPL {X  -156.492, Y  +704.774, Z    +0.000, E1  +414.365, E3 -292612.660}
SPL {X  -154.917, Y  +711.470, Z    +0.000, E1  +414.052, E3 -292624.320}
SPL {X  -153.204, Y  +717.603, Z    +0.000, E1  +413.775, E3 -292635.166}
SPL {X  -151.355, Y  +723.351, Z    +0.000, E1  +413.415, E3 -292645.637}
SPL {X  -148.967, Y  +729.859, Z    +0.000, E1  +413.026, E3 -292657.650}
SPL {X  -145.862, Y  +737.236, Z    +0.000, E1  +412.427, E3 -292671.704}
SPL {X  -142.777, Y  +743.691, Z    +0.000, E1  +411.831, E3 -292684.247}
SPL {X  -132.301, Y  +761.463, Z    +0.000, E1  +405.510, E3 -292763.532}
ENDSPLINE

SPLINE
SPL {X  -145.877, Y  +737.201, Z    +0.000, E1  +394.468, E3 -292846.643}
SPL {X  -152.550, Y  +719.721, Z    +0.000, E1  +387.728, E3 -292862.132}
SPL {X  -157.145, Y  +701.536, Z    +0.000, E1  +379.368, E3 -292871.587}
SPL {X  -159.035, Y  +688.952, Z    +0.000, E1  +372.676, E3 -292875.628}
SPL {X  -159.756, Y  +680.154, Z    +0.000, E1  +367.520, E3 -292877.354}
SPL {X  -159.986, Y  +672.560, Z    +0.000, E1  +362.636, E3 -292878.252}
SPL {X  -159.990, Y  +668.344, Z    +0.000, E1  +359.382, E3 -292878.518}
SPL {X  -159.990, Y  +664.070, Z    +0.000, E1  +354.975, E3 -292878.847}
SPL {X  -159.990, Y  +656.953, Z    +0.000, E1  +346.040, E3 -292879.913}
SPL {X  -159.990, Y  +644.589, Z    +0.000, E1  +330.989, E3 -292883.325}
SPL {X  -159.990, Y  +605.095, Z    +0.000, E1  +310.486, E3 -292908.416}
SPL {X  -159.990, Y  +546.155, Z    +0.000, E1  +305.539, E3 -292971.174}
SPL {X  -159.990, Y  +539.348, Z    +0.000, E1  +305.531, E3 -292981.478}
SPL {X  -159.990, Y  +530.752, Z    +0.000, E1  +305.518, E3 -292994.485}
SPL {X  -159.990, Y  +522.797, Z    +0.000, E1  +305.537, E3 -293006.568}
SPL {X  -159.990, Y  +515.332, Z    +0.000, E1  +305.526, E3 -293017.857}
SPL {X  -159.990, Y  +508.047, Z    +0.000, E1  +305.531, E3 -293028.874}
SPL {X  -159.990, Y  +499.403, Z    +0.000, E1  +305.488, E3 -293041.913}
SPL {X  -159.990, Y  +479.413, Z    +0.000, E1  +302.719, E3 -293053.059}
SPL {X  -159.990, Y  +454.926, Z    +0.000, E1  +299.433, E3 -293062.165}
SPL {X  -159.990, Y  +449.697, Z    +0.000, E1  +300.191, E3 -293073.628}
SPL {X  -159.990, Y  +444.026, Z    +0.000, E1  +301.072, E3 -293086.886}
SPL {X  -159.990, Y  +437.596, Z    +0.000, E1  +301.764, E3 -293099.627}
SPL {X  -159.990, Y  +432.883, Z    +0.000, E1  +302.386, E3 -293110.024}
SPL {X  -159.990, Y  +429.044, Z    +0.000, E1  +303.109, E3 -293119.914}
SPL {X  -159.990, Y  +425.222, Z    +0.000, E1  +304.101, E3 -293131.811}
SPL {X  -159.990, Y  +420.083, Z    +0.000, E1  +304.918, E3 -293144.387}
SPL {X  -159.990, Y  +412.567, Z    +0.000, E1  +305.072, E3 -293156.612}
SPL {X  -159.990, Y  +402.790, Z    +0.000, E1  +305.070, E3 -293171.205}
SPL {X  -159.990, Y  +392.953, Z    +0.000, E1  +305.082, E3 -293185.899}
SPL {X  -159.990, Y  +383.354, Z    +0.000, E1  +305.080, E3 -293200.209}
SPL {X  -159.786, Y  +374.425, Z    +0.000, E1  +305.121, E3 -293213.738}
SPL {X  -159.184, Y  +366.462, Z    +0.000, E1  +305.220, E3 -293226.239}
SPL {X  -158.166, Y  +358.413, Z    +0.000, E1  +305.386, E3 -293239.295}
SPL {X  -156.775, Y  +350.586, Z    +0.000, E1  +305.627, E3 -293252.419}
SPL {X  -155.397, Y  +344.442, Z    +0.000, E1  +305.886, E3 -293263.035}
SPL {X  -153.976, Y  +339.046, Z    +0.000, E1  +306.128, E3 -293272.527}
SPL {X  -152.417, Y  +333.859, Z    +0.000, E1  +306.416, E3 -293281.853}
SPL {X  -150.681, Y  +328.723, Z    +0.000, E1  +306.710, E3 -293291.229}
SPL {X  -147.884, Y  +321.449, Z    +0.000, E1  +307.200, E3 -293304.802}
SPL {X  -145.161, Y  +315.232, Z    +0.000, E1  +307.745, E3 -293316.734}
SPL {X  -142.534, Y  +309.830, Z    +0.000, E1  +308.237, E3 -293327.239}
SPL {X  -132.342, Y  +292.599, Z    +0.000, E1  +315.826, E3 -293424.527}
ENDSPLINE

SPLINE
SPL {X  -151.238, Y  +330.309, Z    +0.000, E1  +330.693, E3 -293497.684}
SPL {X  -156.949, Y  +351.453, Z    +0.000, E1  +340.161, E3 -293509.844}
SPL {X  -159.024, Y  +364.945, Z    +0.000, E1  +347.297, E3 -293514.262}
SPL {X  -159.878, Y  +376.512, Z    +0.000, E1  +354.071, E3 -293516.514}
SPL {X  -159.990, Y  +383.659, Z    +0.000, E1  +358.950, E3 -293517.208}
SPL {X  -159.990, Y  +387.327, Z    +0.000, E1  +362.137, E3 -293517.441}
SPL {X  -159.990, Y  +390.622, Z    +0.000, E1  +365.876, E3 -293517.734}
SPL {X  -159.990, Y  +394.493, Z    +0.000, E1  +370.512, E3 -293518.257}
SPL {X  -159.990, Y  +401.377, Z    +0.000, E1  +379.398, E3 -293519.712}
SPL {X  -159.990, Y  +411.365, Z    +0.000, E1  +390.630, E3 -293522.920}
SPL {X  -159.990, Y  +450.467, Z    +0.000, E1  +410.183, E3 -293546.569}
SPL {X  -159.990, Y  +509.934, Z    +0.000, E1  +414.923, E3 -293609.188}
SPL {X  -159.990, Y  +516.848, Z    +0.000, E1  +414.930, E3 -293619.476}
SPL {X  -159.990, Y  +524.818, Z    +0.000, E1  +414.933, E3 -293631.348}
SPL {X  -159.990, Y  +532.100, Z    +0.000, E1  +414.924, E3 -293642.201}
SPL {X  -159.990, Y  +539.391, Z    +0.000, E1  +414.933, E3 -293653.053}
SPL {X  -159.990, Y  +546.283, Z    +0.000, E1  +414.924, E3 -293663.325}
SPL {X  -159.990, Y  +553.734, Z    +0.000, E1  +414.938, E3 -293674.411}
SPL {X  -159.990, Y  +564.956, Z    +0.000, E1  +414.973, E3 -293691.083}
SPL {X  -159.990, Y  +577.902, Z    +0.000, E1  +414.969, E3 -293710.373}
SPL {X  -159.990, Y  +588.063, Z    +0.000, E1  +414.931, E3 -293725.563}
SPL {X  -159.990, Y  +595.273, Z    +0.000, E1  +414.928, E3 -293736.287}
SPL {X  -159.990, Y  +602.326, Z    +0.000, E1  +414.932, E3 -293746.787}
SPL {X  -159.990, Y  +609.708, Z    +0.000, E1  +414.930, E3 -293757.794}
SPL {X  -159.990, Y  +618.088, Z    +0.000, E1  +414.948, E3 -293770.223}
SPL {X  -159.990, Y  +625.928, Z    +0.000, E1  +414.931, E3 -293781.919}
SPL {X  -159.990, Y  +635.803, Z    +0.000, E1  +414.980, E3 -293796.547}
SPL {X  -159.990, Y  +646.303, Z    +0.000, E1  +414.946, E3 -293812.217}
SPL {X  -159.990, Y  +653.312, Z    +0.000, E1  +414.932, E3 -293822.669}
SPL {X  -159.990, Y  +661.828, Z    +0.000, E1  +414.965, E3 -293835.325}
SPL {X  -159.989, Y  +672.128, Z    +0.000, E1  +414.946, E3 -293850.714}
SPL {X  -159.636, Y  +682.136, Z    +0.000, E1  +414.901, E3 -293865.972}
SPL {X  -158.805, Y  +690.934, Z    +0.000, E1  +414.742, E3 -293879.982}
SPL {X  -157.890, Y  +697.337, Z    +0.000, E1  +414.571, E3 -293890.504}
SPL {X  -156.492, Y  +704.774, Z    +0.000, E1  +414.365, E3 -293902.983}
SPL {X  -154.917, Y  +711.470, Z    +0.000, E1  +414.052, E3 -293914.643}
SPL {X  -153.561, Y  +716.398, Z    +0.000, E1  +413.816, E3 -293923.364}
SPL {X  -151.715, Y  +722.287, Z    +0.000, E1  +413.503, E3 -293933.980}
SPL {X  -149.700, Y  +727.952, Z    +0.000, E1  +413.118, E3 -293944.454}
SPL {X  -147.376, Y  +733.767, Z    +0.000, E1  +412.706, E3 -293955.405}
SPL {X  -145.109, Y  +738.881, Z    +0.000, E1  +412.243, E3 -293965.251}
SPL {X  -142.777, Y  +743.691, Z    +0.000, E1  +411.831, E3 -293974.570}
SPL {X  -132.301, Y  +761.463, Z    +0.000, E1  +405.510, E3 -294053.855}
ENDSPLINE

SPLINE
SPL {X  -145.877, Y  +737.201, Z    +0.000, E1  +394.468, E3 -294136.966}
SPL {X  -152.550, Y  +719.721, Z    +0.000, E1  +387.728, E3 -294152.455}
SPL {X  -157.145, Y  +701.536, Z    +0.000, E1  +379.368, E3 -294161.909}
SPL {X  -159.035, Y  +688.952, Z    +0.000, E1  +372.676, E3 -294165.950}
SPL {X  -159.873, Y  +677.622, Z    +0.000, E1  +366.008, E3 -294168.022}
SPL {X  -159.990, Y  +670.381, Z    +0.000, E1  +361.064, E3 -294168.723}
SPL {X  -159.990, Y  +666.603, Z    +0.000, E1  +357.744, E3 -294168.954}
SPL {X  -159.990, Y  +662.759, Z    +0.000, E1  +353.275, E3 -294169.297}
SPL {X  -159.990, Y  +658.737, Z    +0.000, E1  +348.199, E3 -294169.876}
SPL {X  -159.990, Y  +652.023, Z    +0.000, E1  +339.551, E3 -294171.360}
SPL {X  -159.990, Y  +641.935, Z    +0.000, E1  +328.152, E3 -294174.532}
SPL {X  -159.990, Y  +605.095, Z    +0.000, E1  +310.486, E3 -294198.738}
SPL {X  -159.990, Y  +546.155, Z    +0.000, E1  +305.539, E3 -294261.497}
SPL {X  -159.990, Y  +539.348, Z    +0.000, E1  +305.531, E3 -294271.801}
SPL {X  -159.990, Y  +530.752, Z    +0.000, E1  +305.518, E3 -294284.808}
SPL {X  -159.990, Y  +522.797, Z    +0.000, E1  +305.537, E3 -294296.891}
SPL {X  -159.990, Y  +515.332, Z    +0.000, E1  +305.526, E3 -294308.180}
SPL {X  -159.990, Y  +508.047, Z    +0.000, E1  +305.531, E3 -294319.197}
SPL {X  -159.990, Y  +499.403, Z    +0.000, E1  +305.488, E3 -294332.236}
SPL {X  -159.990, Y  +479.413, Z    +0.000, E1  +302.719, E3 -294343.381}
SPL {X  -159.990, Y  +454.926, Z    +0.000, E1  +299.433, E3 -294352.488}
SPL {X  -159.990, Y  +449.697, Z    +0.000, E1  +300.191, E3 -294363.950}
SPL {X  -159.990, Y  +444.026, Z    +0.000, E1  +301.072, E3 -294377.208}
SPL {X  -159.990, Y  +437.596, Z    +0.000, E1  +301.764, E3 -294389.950}
SPL {X  -159.990, Y  +432.883, Z    +0.000, E1  +302.386, E3 -294400.347}
SPL {X  -159.990, Y  +429.044, Z    +0.000, E1  +303.109, E3 -294410.237}
SPL {X  -159.990, Y  +425.222, Z    +0.000, E1  +304.101, E3 -294422.134}
SPL {X  -159.990, Y  +418.562, Z    +0.000, E1  +304.950, E3 -294437.292}
SPL {X  -159.990, Y  +407.911, Z    +0.000, E1  +305.062, E3 -294453.883}
SPL {X  -159.990, Y  +400.284, Z    +0.000, E1  +305.103, E3 -294465.317}
SPL {X  -159.990, Y  +392.953, Z    +0.000, E1  +305.082, E3 -294476.222}
SPL {X  -159.990, Y  +383.354, Z    +0.000, E1  +305.080, E3 -294490.532}
SPL {X  -159.786, Y  +374.425, Z    +0.000, E1  +305.121, E3 -294504.061}
SPL {X  -159.184, Y  +366.462, Z    +0.000, E1  +305.220, E3 -294516.561}
SPL {X  -158.166, Y  +358.413, Z    +0.000, E1  +305.386, E3 -294529.617}
SPL {X  -156.775, Y  +350.586, Z    +0.000, E1  +305.627, E3 -294542.742}
SPL {X  -155.397, Y  +344.442, Z    +0.000, E1  +305.886, E3 -294553.357}
SPL {X  -153.976, Y  +339.046, Z    +0.000, E1  +306.128, E3 -294562.849}
SPL {X  -152.417, Y  +333.859, Z    +0.000, E1  +306.416, E3 -294572.176}
SPL {X  -150.681, Y  +328.723, Z    +0.000, E1  +306.710, E3 -294581.552}
SPL {X  -147.884, Y  +321.449, Z    +0.000, E1  +307.200, E3 -294595.125}
SPL {X  -145.161, Y  +315.232, Z    +0.000, E1  +307.745, E3 -294607.056}
SPL {X  -142.534, Y  +309.830, Z    +0.000, E1  +308.237, E3 -294617.561}
SPL {X  -132.342, Y  +292.599, Z    +0.000, E1  +315.826, E3 -294714.849}
ENDSPLINE

SPLINE
SPL {X  -151.238, Y  +330.309, Z    +0.000, E1  +330.693, E3 -294788.006}
SPL {X  -156.949, Y  +351.453, Z    +0.000, E1  +340.161, E3 -294800.167}
SPL {X  -159.024, Y  +364.945, Z    +0.000, E1  +347.297, E3 -294804.585}
SPL {X  -159.758, Y  +373.891, Z    +0.000, E1  +352.513, E3 -294806.473}
SPL {X  -159.985, Y  +381.208, Z    +0.000, E1  +357.184, E3 -294807.356}
SPL {X  -159.990, Y  +384.493, Z    +0.000, E1  +359.676, E3 -294807.581}
SPL {X  -159.990, Y  +387.327, Z    +0.000, E1  +362.137, E3 -294807.764}
SPL {X  -159.990, Y  +392.053, Z    +0.000, E1  +367.477, E3 -294808.229}
SPL {X  -159.990, Y  +396.158, Z    +0.000, E1  +372.775, E3 -294808.854}
SPL {X  -159.990, Y  +401.377, Z    +0.000, E1  +379.398, E3 -294810.035}
SPL {X  -159.990, Y  +411.365, Z    +0.000, E1  +390.630, E3 -294813.243}
SPL {X  -159.990, Y  +450.467, Z    +0.000, E1  +410.183, E3 -294836.892}
SPL {X  -159.990, Y  +509.934, Z    +0.000, E1  +414.923, E3 -294899.511}
SPL {X  -159.990, Y  +516.848, Z    +0.000, E1  +414.930, E3 -294909.799}
SPL {X  -159.990, Y  +524.818, Z    +0.000, E1  +414.933, E3 -294921.671}
SPL {X  -159.990, Y  +532.100, Z    +0.000, E1  +414.924, E3 -294932.524}
SPL {X  -159.990, Y  +539.391, Z    +0.000, E1  +414.933, E3 -294943.376}
SPL {X  -159.990, Y  +546.283, Z    +0.000, E1  +414.924, E3 -294953.647}
SPL {X  -159.990, Y  +553.734, Z    +0.000, E1  +414.938, E3 -294964.734}
SPL {X  -159.990, Y  +564.956, Z    +0.000, E1  +414.973, E3 -294981.405}
SPL {X  -159.990, Y  +577.902, Z    +0.000, E1  +414.969, E3 -295000.695}
SPL {X  -159.990, Y  +588.063, Z    +0.000, E1  +414.931, E3 -295015.886}
SPL {X  -159.990, Y  +595.273, Z    +0.000, E1  +414.928, E3 -295026.610}
SPL {X  -159.990, Y  +602.326, Z    +0.000, E1  +414.932, E3 -295037.110}
SPL {X  -159.990, Y  +609.708, Z    +0.000, E1  +414.930, E3 -295048.117}
SPL {X  -159.990, Y  +618.088, Z    +0.000, E1  +414.948, E3 -295060.545}
SPL {X  -159.990, Y  +625.928, Z    +0.000, E1  +414.931, E3 -295072.241}
SPL {X  -159.990, Y  +635.803, Z    +0.000, E1  +414.980, E3 -295086.869}
SPL {X  -159.990, Y  +646.303, Z    +0.000, E1  +414.946, E3 -295102.540}
SPL {X  -159.990, Y  +656.335, Z    +0.000, E1  +414.969, E3 -295117.442}
SPL {X  -159.990, Y  +664.577, Z    +0.000, E1  +414.924, E3 -295129.820}
SPL {X  -159.989, Y  +672.128, Z    +0.000, E1  +414.946, E3 -295141.036}
SPL {X  -159.792, Y  +679.466, Z    +0.000, E1  +414.893, E3 -295152.194}
SPL {X  -159.330, Y  +686.016, Z    +0.000, E1  +414.837, E3 -295162.425}
SPL {X  -158.190, Y  +695.432, Z    +0.000, E1  +414.658, E3 -295177.622}
SPL {X  -157.027, Y  +702.151, Z    +0.000, E1  +414.415, E3 -295188.904}
SPL {X  -156.112, Y  +706.513, Z    +0.000, E1  +414.265, E3 -295196.338}
SPL {X  -154.917, Y  +711.470, Z    +0.000, E1  +414.052, E3 -295204.965}
SPL {X  -153.561, Y  +716.398, Z    +0.000, E1  +413.816, E3 -295213.687}
SPL {X  -151.715, Y  +722.287, Z    +0.000, E1  +413.503, E3 -295224.303}
SPL {X  -149.700, Y  +727.952, Z    +0.000, E1  +413.118, E3 -295234.777}
SPL {X  -147.376, Y  +733.767, Z    +0.000, E1  +412.706, E3 -295245.727}
SPL {X  -145.109, Y  +738.881, Z    +0.000, E1  +412.243, E3 -295255.574}
SPL {X  -142.777, Y  +743.691, Z    +0.000, E1  +411.831, E3 -295264.892}
SPL {X  -132.301, Y  +761.463, Z    +0.000, E1  +405.510, E3 -295344.177}
ENDSPLINE

SPLINE
SPL {X  -145.877, Y  +737.201, Z    +0.000, E1  +394.468, E3 -295427.288}
SPL {X  -152.550, Y  +719.721, Z    +0.000, E1  +387.728, E3 -295442.777}
SPL {X  -157.145, Y  +701.536, Z    +0.000, E1  +379.368, E3 -295452.232}
SPL {X  -159.035, Y  +688.952, Z    +0.000, E1  +372.676, E3 -295456.273}
SPL {X  -159.756, Y  +680.154, Z    +0.000, E1  +367.520, E3 -295457.999}
SPL {X  -159.986, Y  +672.560, Z    +0.000, E1  +362.636, E3 -295458.897}
SPL {X  -159.990, Y  +669.364, Z    +0.000, E1  +360.170, E3 -295459.105}
SPL {X  -159.990, Y  +666.603, Z    +0.000, E1  +357.744, E3 -295459.277}
SPL {X  -159.990, Y  +662.759, Z    +0.000, E1  +353.275, E3 -295459.620}
SPL {X  -159.990, Y  +658.737, Z    +0.000, E1  +348.199, E3 -295460.198}
SPL {X  -159.990, Y  +652.023, Z    +0.000, E1  +339.551, E3 -295461.682}
SPL {X  -159.990, Y  +641.935, Z    +0.000, E1  +328.152, E3 -295464.854}
SPL {X  -159.990, Y  +605.095, Z    +0.000, E1  +310.486, E3 -295489.061}
SPL {X  -159.990, Y  +546.155, Z    +0.000, E1  +305.539, E3 -295551.819}
SPL {X  -159.990, Y  +539.348, Z    +0.000, E1  +305.531, E3 -295562.123}
SPL {X  -159.990, Y  +530.752, Z    +0.000, E1  +305.518, E3 -295575.131}
SPL {X  -159.990, Y  +522.797, Z    +0.000, E1  +305.537, E3 -295587.214}
SPL {X  -159.990, Y  +515.332, Z    +0.000, E1  +305.526, E3 -295598.503}
SPL {X  -159.990, Y  +508.047, Z    +0.000, E1  +305.531, E3 -295609.519}
SPL {X  -159.990, Y  +501.296, Z    +0.000, E1  +305.518, E3 -295619.741}
SPL {X  -159.990, Y  +487.558, Z    +0.000, E1  +304.151, E3 -295631.371}
SPL {X  -159.990, Y  +454.926, Z    +0.000, E1  +299.433, E3 -295642.810}
SPL {X  -159.990, Y  +449.697, Z    +0.000, E1  +300.191, E3 -295654.273}
SPL {X  -159.990, Y  +445.847, Z    +0.000, E1  +300.905, E3 -295663.896}
SPL {X  -159.990, Y  +439.266, Z    +0.000, E1  +301.568, E3 -295676.979}
SPL {X  -159.990, Y  +432.883, Z    +0.000, E1  +302.386, E3 -295690.669}
SPL {X  -159.990, Y  +429.044, Z    +0.000, E1  +303.109, E3 -295700.560}
SPL {X  -159.990, Y  +425.222, Z    +0.000, E1  +304.101, E3 -295712.457}
SPL {X  -159.990, Y  +420.083, Z    +0.000, E1  +304.918, E3 -295725.033}
ENDSPLINE

SPLINE
SPL {X  -159.990, Y  +436.353, Z    +0.000, E1  +311.446, E3 -295738.215}
ENDSPLINE

SPLINE
SPL {X  -159.990, Y  +429.614, Z    +0.000, E1  +311.486, E3 -295750.935}
SPL {X  -159.990, Y  +423.677, Z    +0.000, E1  +311.471, E3 -295762.047}
SPL {X  -159.990, Y  +417.714, Z    +0.000, E1  +311.484, E3 -295773.257}
SPL {X  -159.990, Y  +412.449, Z    +0.000, E1  +311.483, E3 -295783.117}
SPL {X  -159.990, Y  +406.256, Z    +0.000, E1  +311.459, E3 -295794.685}
SPL {X  -159.990, Y  +399.971, Z    +0.000, E1  +311.480, E3 -295806.500}
SPL {X  -159.990, Y  +394.711, Z    +0.000, E1  +311.476, E3 -295816.358}
SPL {X  -159.990, Y  +387.710, Z    +0.000, E1  +311.455, E3 -295829.481}
SPL {X  -159.984, Y  +381.116, Z    +0.000, E1  +311.484, E3 -295841.898}
SPL {X  -159.797, Y  +374.648, Z    +0.000, E1  +311.491, E3 -295854.193}
SPL {X  -159.230, Y  +366.920, Z    +0.000, E1  +311.592, E3 -295869.293}
SPL {X  -158.297, Y  +359.284, Z    +0.000, E1  +311.753, E3 -295884.592}
SPL {X  -157.042, Y  +351.926, Z    +0.000, E1  +311.986, E3 -295899.715}
SPL {X  -155.408, Y  +344.485, Z    +0.000, E1  +312.267, E3 -295915.344}
SPL {X  -153.753, Y  +338.264, Z    +0.000, E1  +312.613, E3 -295928.773}
SPL {X  -152.142, Y  +333.005, Z    +0.000, E1  +312.891, E3 -295940.247}
SPL {X  -150.309, Y  +327.691, Z    +0.000, E1  +313.264, E3 -295952.102}
SPL {X  -148.834, Y  +323.804, Z    +0.000, E1  +313.556, E3 -295960.865}
SPL {X  -147.343, Y  +320.157, Z    +0.000, E1  +313.838, E3 -295969.155}
SPL {X  -142.380, Y  +309.529, Z    +0.000, E1  +319.953, E3 -296041.915}
ENDSPLINE

SPLINE
SPL {X  -153.420, Y  +337.122, Z    +0.000, E1  +333.501, E3 -296099.413}
SPL {X  -157.288, Y  +353.220, Z    +0.000, E1  +341.134, E3 -296111.459}
SPL {X  -159.049, Y  +365.172, Z    +0.000, E1  +347.392, E3 -296117.012}
SPL {X  -159.881, Y  +376.607, Z    +0.000, E1  +353.914, E3 -296120.241}
SPL {X  -159.990, Y  +384.736, Z    +0.000, E1  +359.276, E3 -296121.492}
SPL {X  -159.990, Y  +388.564, Z    +0.000, E1  +362.561, E3 -296121.956}
SPL {X  -159.990, Y  +392.444, Z    +0.000, E1  +366.277, E3 -296122.577}
SPL {X  -159.990, Y  +398.585, Z    +0.000, E1  +372.930, E3 -296123.957}
SPL {X  -159.990, Y  +408.423, Z    +0.000, E1  +383.302, E3 -296127.491}
SPL {X  -159.990, Y  +438.418, Z    +0.000, E1  +401.067, E3 -296149.064}
SPL {X  -159.990, Y  +482.913, Z    +0.000, E1  +407.036, E3 -296208.419}
SPL {X  -159.990, Y  +489.230, Z    +0.000, E1  +407.019, E3 -296220.930}
SPL {X  -159.990, Y  +495.241, Z    +0.000, E1  +407.026, E3 -296232.809}
SPL {X  -159.990, Y  +501.001, Z    +0.000, E1  +407.020, E3 -296244.186}
SPL {X  -159.990, Y  +506.758, Z    +0.000, E1  +407.038, E3 -296255.532}
SPL {X  -159.990, Y  +512.807, Z    +0.000, E1  +407.022, E3 -296267.523}
SPL {X  -159.990, Y  +518.043, Z    +0.000, E1  +407.016, E3 -296277.901}
SPL {X  -159.990, Y  +523.058, Z    +0.000, E1  +407.015, E3 -296287.817}
SPL {X  -159.990, Y  +527.746, Z    +0.000, E1  +407.012, E3 -296297.090}
SPL {X  -159.990, Y  +533.771, Z    +0.000, E1  +407.034, E3 -296308.975}
SPL {X  -159.990, Y  +542.379, Z    +0.000, E1  +407.067, E3 -296325.945}
SPL {X  -159.990, Y  +549.846, Z    +0.000, E1  +407.016, E3 -296340.790}
SPL {X  -159.990, Y  +554.843, Z    +0.000, E1  +407.014, E3 -296350.668}
SPL {X  -159.990, Y  +560.453, Z    +0.000, E1  +407.023, E3 -296361.751}
SPL {X  -159.990, Y  +566.612, Z    +0.000, E1  +407.022, E3 -296373.933}
SPL {X  -159.990, Y  +572.901, Z    +0.000, E1  +407.028, E3 -296386.345}
SPL {X  -159.990, Y  +578.640, Z    +0.000, E1  +407.021, E3 -296397.697}
SPL {X  -159.990, Y  +583.515, Z    +0.000, E1  +407.019, E3 -296407.336}
SPL {X  -159.990, Y  +589.675, Z    +0.000, E1  +407.042, E3 -296419.474}
SPL {X  -159.990, Y  +596.627, Z    +0.000, E1  +407.034, E3 -296433.214}
SPL {X  -159.990, Y  +602.039, Z    +0.000, E1  +407.021, E3 -296443.921}
SPL {X  -159.990, Y  +607.106, Z    +0.000, E1  +407.028, E3 -296453.928}
SPL {X  -159.990, Y  +612.418, Z    +0.000, E1  +407.023, E3 -296464.440}
SPL {X  -159.990, Y  +618.496, Z    +0.000, E1  +407.049, E3 -296476.406}
SPL {X  -159.990, Y  +624.357, Z    +0.000, E1  +407.020, E3 -296488.032}
SPL {X  -159.990, Y  +629.711, Z    +0.000, E1  +407.034, E3 -296498.601}
SPL {X  -159.990, Y  +635.041, Z    +0.000, E1  +407.022, E3 -296509.146}
SPL {X  -159.990, Y  +639.998, Z    +0.000, E1  +407.027, E3 -296518.938}
SPL {X  -159.990, Y  +646.188, Z    +0.000, E1  +407.041, E3 -296531.164}
SPL {X  -159.990, Y  +652.067, Z    +0.000, E1  +407.023, E3 -296542.800}
SPL {X  -159.990, Y  +657.109, Z    +0.000, E1  +407.025, E3 -296552.779}
SPL {X  -159.990, Y  +662.651, Z    +0.000, E1  +407.027, E3 -296563.735}
SPL {X  -159.990, Y  +668.015, Z    +0.000, E1  +407.025, E3 -296574.335}
SPL {X  -159.972, Y  +673.909, Z    +0.000, E1  +407.029, E3 -296586.001}
SPL {X  -159.776, Y  +679.772, Z    +0.000, E1  +406.992, E3 -296597.802}
SPL {X  -159.384, Y  +685.411, Z    +0.000, E1  +406.921, E3 -296609.363}
SPL {X  -158.642, Y  +692.228, Z    +0.000, E1  +406.819, E3 -296623.578}
SPL {X  -157.651, Y  +698.760, Z    +0.000, E1  +406.609, E3 -296637.573}
SPL {X  -156.719, Y  +703.686, Z    +0.000, E1  +406.438, E3 -296648.266}
SPL {X  -155.778, Y  +707.970, Z    +0.000, E1  +406.262, E3 -296657.741}
SPL {X  -154.419, Y  +713.351, Z    +0.000, E1  +406.025, E3 -296669.772}
SPL {X  -152.913, Y  +718.557, Z    +0.000, E1  +405.729, E3 -296681.624}
SPL {X  -151.262, Y  +723.621, Z    +0.000, E1  +405.429, E3 -296693.290}
SPL {X  -149.074, Y  +729.584, Z    +0.000, E1  +405.040, E3 -296707.219}
SPL {X  -142.577, Y  +744.086, Z    +0.000, E1  +400.686, E3 -296773.425}
ENDSPLINE

SPLINE
SPL {X  -152.566, Y  +719.671, Z    +0.000, E1  +387.682, E3 -296843.896}
SPL {X  -158.253, Y  +695.011, Z    +0.000, E1  +375.913, E3 -296860.568}
SPL {X  -159.486, Y  +684.192, Z    +0.000, E1  +369.965, E3 -296864.514}
SPL {X  -159.898, Y  +676.924, Z    +0.000, E1  +365.683, E3 -296866.212}
SPL {X  -159.990, Y  +671.720, Z    +0.000, E1  +362.298, E3 -296867.052}
SPL {X  -159.990, Y  +668.164, Z    +0.000, E1  +359.695, E3 -296867.468}
SPL {X  -159.990, Y  +665.062, Z    +0.000, E1  +356.961, E3 -296867.807}
SPL {X  -159.990, Y  +660.795, Z    +0.000, E1  +352.651, E3 -296868.470}
SPL {X  -159.990, Y  +654.574, Z    +0.000, E1  +345.673, E3 -296869.925}
SPL {X  -159.990, Y  +647.816, Z    +0.000, E1  +338.252, E3 -296872.176}
SPL {X  -159.990, Y  +640.751, Z    +0.000, E1  +331.747, E3 -296875.770}
SPL {X  -159.990, Y  +611.706, Z    +0.000, E1  +317.244, E3 -296898.543}
SPL {X  -159.990, Y  +567.814, Z    +0.000, E1  +312.360, E3 -296958.633}
SPL {X  -159.990, Y  +558.774, Z    +0.000, E1  +312.384, E3 -296976.199}
SPL {X  -159.990, Y  +550.551, Z    +0.000, E1  +312.385, E3 -296992.140}
SPL {X  -159.990, Y  +542.502, Z    +0.000, E1  +312.392, E3 -297007.755}
SPL {X  -159.990, Y  +536.986, Z    +0.000, E1  +312.423, E3 -297018.475}
SPL {X  -159.990, Y  +532.938, Z    +0.000, E1  +312.415, E3 -297026.301}
SPL {X  -159.990, Y  +525.893, Z    +0.000, E1  +312.375, E3 -297039.915}
SPL {X  -159.990, Y  +518.864, Z    +0.000, E1  +312.415, E3 -297053.597}
SPL {X  -159.990, Y  +512.328, Z    +0.000, E1  +312.388, E3 -297066.231}
SPL {X  -159.990, Y  +505.755, Z    +0.000, E1  +312.413, E3 -297079.008}
ENDSPLINE

SPLINE
SPL {X  -159.990, Y  +517.758, Z    +0.000, E1  +318.109, E3 -297086.731}
ENDSPLINE

SPLINE
SPL {X  -159.990, Y  +516.975, Z    +0.000, E1  +319.588, E3 -297097.795}
SPL {X  -159.990, Y  +508.583, Z    +0.000, E1  +318.552, E3 -297112.100}
SPL {X  -159.990, Y  +499.983, Z    +0.000, E1  +317.561, E3 -297126.554}
SPL {X  -159.990, Y  +492.624, Z    +0.000, E1  +316.776, E3 -297138.658}
SPL {X  -159.990, Y  +485.551, Z    +0.000, E1  +316.053, E3 -297150.208}
SPL {X  -159.990, Y  +477.585, Z    +0.000, E1  +315.156, E3 -297162.118}
SPL {X  -159.990, Y  +470.785, Z    +0.000, E1  +314.453, E3 -297172.291}
SPL {X  -159.990, Y  +463.371, Z    +0.000, E1  +313.690, E3 -297183.016}
SPL {X  -159.990, Y  +455.469, Z    +0.000, E1  +312.807, E3 -297193.542}
SPL {X  -159.990, Y  +445.848, Z    +0.000, E1  +311.866, E3 -297206.634}
SPL {X  -159.990, Y  +436.400, Z    +0.000, E1  +311.449, E3 -297222.016}
SPL {X  -159.990, Y  +429.614, Z    +0.000, E1  +311.486, E3 -297234.806}
SPL {X  -159.990, Y  +423.677, Z    +0.000, E1  +311.471, E3 -297245.918}
SPL {X  -159.990, Y  +417.714, Z    +0.000, E1  +311.484, E3 -297257.128}
SPL {X  -159.990, Y  +412.449, Z    +0.000, E1  +311.483, E3 -297266.988}
SPL {X  -159.990, Y  +406.256, Z    +0.000, E1  +311.459, E3 -297278.556}
SPL {X  -159.990, Y  +399.971, Z    +0.000, E1  +311.480, E3 -297290.371}
SPL {X  -159.990, Y  +394.711, Z    +0.000, E1  +311.476, E3 -297300.229}
SPL {X  -159.990, Y  +387.710, Z    +0.000, E1  +311.455, E3 -297313.352}
SPL {X  -159.966, Y  +379.751, Z    +0.000, E1  +311.465, E3 -297328.316}
SPL {X  -159.734, Y  +373.449, Z    +0.000, E1  +311.528, E3 -297340.420}
SPL {X  -159.230, Y  +366.920, Z    +0.000, E1  +311.592, E3 -297353.164}
SPL {X  -158.532, Y  +360.951, Z    +0.000, E1  +311.745, E3 -297365.137}
SPL {X  -157.692, Y  +355.479, Z    +0.000, E1  +311.882, E3 -297376.265}
SPL {X  -156.349, Y  +348.560, Z    +0.000, E1  +312.101, E3 -297390.604}
SPL {X  -154.984, Y  +342.790, Z    +0.000, E1  +312.392, E3 -297402.901}
SPL {X  -153.247, Y  +336.540, Z    +0.000, E1  +312.660, E3 -297416.337}
SPL {X  -150.765, Y  +328.959, Z    +0.000, E1  +313.136, E3 -297433.083}
SPL {X  -148.834, Y  +323.804, Z    +0.000, E1  +313.556, E3 -297444.736}
SPL {X  -147.343, Y  +320.157, Z    +0.000, E1  +313.838, E3 -297453.026}
SPL {X  -142.380, Y  +309.529, Z    +0.000, E1  +319.953, E3 -297525.786}
ENDSPLINE

SPLINE
SPL {X  -153.420, Y  +337.122, Z    +0.000, E1  +333.501, E3 -297583.284}
SPL {X  -157.288, Y  +353.220, Z    +0.000, E1  +341.134, E3 -297595.330}
SPL {X  -159.049, Y  +365.172, Z    +0.000, E1  +347.392, E3 -297600.883}
SPL {X  -159.881, Y  +376.607, Z    +0.000, E1  +353.914, E3 -297604.112}
SPL {X  -159.990, Y  +383.110, Z    +0.000, E1  +358.202, E3 -297605.165}
SPL {X  -159.990, Y  +387.352, Z    +0.000, E1  +361.387, E3 -297605.680}
SPL {X  -159.990, Y  +391.188, Z    +0.000, E1  +365.082, E3 -297606.221}
SPL {X  -159.990, Y  +395.106, Z    +0.000, E1  +369.154, E3 -297606.962}
SPL {X  -159.990, Y  +400.303, Z    +0.000, E1  +374.927, E3 -297608.283}
SPL {X  -159.990, Y  +408.423, Z    +0.000, E1  +383.302, E3 -297611.362}
SPL {X  -159.990, Y  +438.418, Z    +0.000, E1  +401.067, E3 -297632.935}
SPL {X  -159.990, Y  +481.123, Z    +0.000, E1  +407.011, E3 -297688.793}
SPL {X  -159.990, Y  +487.829, Z    +0.000, E1  +407.049, E3 -297701.990}
SPL {X  -159.990, Y  +495.241, Z    +0.000, E1  +407.026, E3 -297716.680}
SPL {X  -159.990, Y  +502.770, Z    +0.000, E1  +407.054, E3 -297731.503}
SPL {X  -159.990, Y  +511.332, Z    +0.000, E1  +407.054, E3 -297748.432}
SPL {X  -159.990, Y  +518.043, Z    +0.000, E1  +407.016, E3 -297761.772}
SPL {X  -159.990, Y  +523.058, Z    +0.000, E1  +407.015, E3 -297771.688}
SPL {X  -159.990, Y  +529.544, Z    +0.000, E1  +407.044, E3 -297784.469}
SPL {X  -159.990, Y  +538.402, Z    +0.000, E1  +407.063, E3 -297801.958}
SPL {X  -159.990, Y  +547.787, Z    +0.000, E1  +407.067, E3 -297820.503}
SPL {X  -159.990, Y  +554.843, Z    +0.000, E1  +407.014, E3 -297834.539}
SPL {X  -159.990, Y  +560.453, Z    +0.000, E1  +407.023, E3 -297845.622}
SPL {X  -159.990, Y  +566.612, Z    +0.000, E1  +407.022, E3 -297857.804}
SPL {X  -159.990, Y  +572.901, Z    +0.000, E1  +407.028, E3 -297870.216}
SPL {X  -159.990, Y  +578.640, Z    +0.000, E1  +407.021, E3 -297881.568}
SPL {X  -159.990, Y  +583.515, Z    +0.000, E1  +407.019, E3 -297891.207}
SPL {X  -159.990, Y  +589.675, Z    +0.000, E1  +407.042, E3 -297903.345}
SPL {X  -159.990, Y  +596.627, Z    +0.000, E1  +407.034, E3 -297917.085}
SPL {X  -159.990, Y  +602.039, Z    +0.000, E1  +407.021, E3 -297927.792}
SPL {X  -159.990, Y  +607.106, Z    +0.000, E1  +407.028, E3 -297937.799}
SPL {X  -159.990, Y  +614.483, Z    +0.000, E1  +407.064, E3 -297952.331}
SPL {X  -159.990, Y  +622.758, Z    +0.000, E1  +407.049, E3 -297968.702}
SPL {X  -159.990, Y  +629.711, Z    +0.000, E1  +407.034, E3 -297982.472}
SPL {X  -159.990, Y  +635.041, Z    +0.000, E1  +407.022, E3 -297993.017}
SPL {X  -159.990, Y  +642.261, Z    +0.000, E1  +407.074, E3 -298007.217}
SPL {X  -159.990, Y  +650.752, Z    +0.000, E1  +407.046, E3 -298024.044}
SPL {X  -159.990, Y  +657.109, Z    +0.000, E1  +407.025, E3 -298036.650}
SPL {X  -159.990, Y  +662.651, Z    +0.000, E1  +407.027, E3 -298047.606}
SPL {X  -159.990, Y  +668.015, Z    +0.000, E1  +407.025, E3 -298058.206}
SPL {X  -159.972, Y  +673.909, Z    +0.000, E1  +407.029, E3 -298069.872}
SPL {X  -159.776, Y  +679.772, Z    +0.000, E1  +406.992, E3 -298081.673}
SPL {X  -159.384, Y  +685.411, Z    +0.000, E1  +406.921, E3 -298093.234}
SPL {X  -158.642, Y  +692.228, Z    +0.000, E1  +406.819, E3 -298107.449}
SPL {X  -157.651, Y  +698.760, Z    +0.000, E1  +406.609, E3 -298121.444}
SPL {X  -156.719, Y  +703.686, Z    +0.000, E1  +406.438, E3 -298132.137}
SPL {X  -155.778, Y  +707.970, Z    +0.000, E1  +406.262, E3 -298141.612}
SPL {X  -154.419, Y  +713.351, Z    +0.000, E1  +406.025, E3 -298153.643}
SPL {X  -152.913, Y  +718.557, Z    +0.000, E1  +405.729, E3 -298165.495}
SPL {X  -151.262, Y  +723.621, Z    +0.000, E1  +405.429, E3 -298177.161}
SPL {X  -149.074, Y  +729.584, Z    +0.000, E1  +405.040, E3 -298191.090}
SPL {X  -142.577, Y  +744.086, Z    +0.000, E1  +400.686, E3 -298257.296}
ENDSPLINE

SPLINE
SPL {X  -152.566, Y  +719.671, Z    +0.000, E1  +387.682, E3 -298327.767}
SPL {X  -158.253, Y  +695.011, Z    +0.000, E1  +375.913, E3 -298344.439}
SPL {X  -159.486, Y  +684.192, Z    +0.000, E1  +369.965, E3 -298348.385}
SPL {X  -159.898, Y  +676.924, Z    +0.000, E1  +365.683, E3 -298350.083}
SPL {X  -159.990, Y  +671.720, Z    +0.000, E1  +362.298, E3 -298350.923}
SPL {X  -159.990, Y  +668.164, Z    +0.000, E1  +359.695, E3 -298351.339}
SPL {X  -159.990, Y  +665.062, Z    +0.000, E1  +356.961, E3 -298351.678}
SPL {X  -159.990, Y  +660.795, Z    +0.000, E1  +352.651, E3 -298352.341}
SPL {X  -159.990, Y  +654.574, Z    +0.000, E1  +345.673, E3 -298353.796}
SPL {X  -159.990, Y  +644.002, Z    +0.000, E1  +334.724, E3 -298357.993}
SPL {X  -159.990, Y  +611.706, Z    +0.000, E1  +317.244, E3 -298382.414}
SPL {X  -159.990, Y  +571.318, Z    +0.000, E1  +312.417, E3 -298435.798}
SPL {X  -159.990, Y  +564.395, Z    +0.000, E1  +312.373, E3 -298449.156}
SPL {X  -159.990, Y  +555.871, Z    +0.000, E1  +312.389, E3 -298465.705}
SPL {X  -159.990, Y  +549.223, Z    +0.000, E1  +312.413, E3 -298478.628}
SPL {X  -159.990, Y  +542.502, Z    +0.000, E1  +312.392, E3 -298491.626}
SPL {X  -159.990, Y  +534.538, Z    +0.000, E1  +312.385, E3 -298507.030}
SPL {X  -159.990, Y  +527.222, Z    +0.000, E1  +312.401, E3 -298521.238}
SPL {X  -159.990, Y  +520.237, Z    +0.000, E1  +312.390, E3 -298534.769}
SPL {X  -159.990, Y  +512.328, Z    +0.000, E1  +312.388, E3 -298550.102}
SPL {X  -159.990, Y  +505.755, Z    +0.000, E1  +312.413, E3 -298562.879}
ENDSPLINE

SPLINE
SPL {X  -159.990, Y  +517.758, Z    +0.000, E1  +318.109, E3 -298570.602}
ENDSPLINE

SPLINE
SPL {X  -159.990, Y  +516.975, Z    +0.000, E1  +319.588, E3 -298581.666}
SPL {X  -159.990, Y  +508.583, Z    +0.000, E1  +318.552, E3 -298595.971}
SPL {X  -159.990, Y  +499.983, Z    +0.000, E1  +317.561, E3 -298610.425}
SPL {X  -159.990, Y  +490.062, Z    +0.000, E1  +316.490, E3 -298626.709}
SPL {X  -159.990, Y  +479.678, Z    +0.000, E1  +315.383, E3 -298642.929}
SPL {X  -159.990, Y  +468.709, Z    +0.000, E1  +314.219, E3 -298659.167}
SPL {X  -159.990, Y  +457.446, Z    +0.000, E1  +313.017, E3 -298674.820}
SPL {X  -159.990, Y  +445.848, Z    +0.000, E1  +311.866, E3 -298690.505}
SPL {X  -159.990, Y  +436.400, Z    +0.000, E1  +311.449, E3 -298705.887}
SPL {X  -159.990, Y  +429.614, Z    +0.000, E1  +311.486, E3 -298718.677}
SPL {X  -159.990, Y  +423.677, Z    +0.000, E1  +311.471, E3 -298729.789}
SPL {X  -159.990, Y  +417.714, Z    +0.000, E1  +311.484, E3 -298740.999}
SPL {X  -159.990, Y  +412.449, Z    +0.000, E1  +311.483, E3 -298750.859}
SPL {X  -159.990, Y  +406.256, Z    +0.000, E1  +311.459, E3 -298762.427}
SPL {X  -159.990, Y  +399.971, Z    +0.000, E1  +311.480, E3 -298774.242}
SPL {X  -159.990, Y  +394.711, Z    +0.000, E1  +311.476, E3 -298784.100}
SPL {X  -159.990, Y  +387.710, Z    +0.000, E1  +311.455, E3 -298797.223}
SPL {X  -159.984, Y  +381.116, Z    +0.000, E1  +311.484, E3 -298809.640}
SPL {X  -159.797, Y  +374.648, Z    +0.000, E1  +311.491, E3 -298821.935}
SPL {X  -159.230, Y  +366.920, Z    +0.000, E1  +311.592, E3 -298837.034}
SPL {X  -158.297, Y  +359.284, Z    +0.000, E1  +311.753, E3 -298852.334}
SPL {X  -157.042, Y  +351.926, Z    +0.000, E1  +311.986, E3 -298867.457}
SPL {X  -155.408, Y  +344.485, Z    +0.000, E1  +312.267, E3 -298883.086}
SPL {X  -153.753, Y  +338.264, Z    +0.000, E1  +312.613, E3 -298896.515}
SPL {X  -152.142, Y  +333.005, Z    +0.000, E1  +312.891, E3 -298907.989}
SPL {X  -150.309, Y  +327.691, Z    +0.000, E1  +313.264, E3 -298919.844}
SPL {X  -148.834, Y  +323.804, Z    +0.000, E1  +313.556, E3 -298928.607}
SPL {X  -147.343, Y  +320.157, Z    +0.000, E1  +313.838, E3 -298936.897}
SPL {X  -142.380, Y  +309.529, Z    +0.000, E1  +319.953, E3 -299009.657}
ENDSPLINE

SPLINE
SPL {X  -153.420, Y  +337.122, Z    +0.000, E1  +333.501, E3 -299067.155}
SPL {X  -157.288, Y  +353.220, Z    +0.000, E1  +341.134, E3 -299079.201}
SPL {X  -159.049, Y  +365.172, Z    +0.000, E1  +347.392, E3 -299084.754}
SPL {X  -159.881, Y  +376.607, Z    +0.000, E1  +353.914, E3 -299087.983}
SPL {X  -159.990, Y  +384.736, Z    +0.000, E1  +359.276, E3 -299089.234}
SPL {X  -159.990, Y  +388.564, Z    +0.000, E1  +362.561, E3 -299089.698}
SPL {X  -159.990, Y  +392.444, Z    +0.000, E1  +366.277, E3 -299090.319}
SPL {X  -159.990, Y  +398.585, Z    +0.000, E1  +372.930, E3 -299091.699}
SPL {X  -159.990, Y  +408.423, Z    +0.000, E1  +383.302, E3 -299095.233}
SPL {X  -159.990, Y  +438.418, Z    +0.000, E1  +401.067, E3 -299116.806}
SPL {X  -159.990, Y  +482.913, Z    +0.000, E1  +407.036, E3 -299176.160}
SPL {X  -159.990, Y  +489.230, Z    +0.000, E1  +407.019, E3 -299188.672}
SPL {X  -159.990, Y  +495.241, Z    +0.000, E1  +407.026, E3 -299200.551}
SPL {X  -159.990, Y  +501.001, Z    +0.000, E1  +407.020, E3 -299211.928}
SPL {X  -159.990, Y  +506.758, Z    +0.000, E1  +407.038, E3 -299223.274}
SPL {X  -159.990, Y  +512.807, Z    +0.000, E1  +407.022, E3 -299235.265}
SPL {X  -159.990, Y  +518.043, Z    +0.000, E1  +407.016, E3 -299245.643}
SPL {X  -159.990, Y  +523.058, Z    +0.000, E1  +407.015, E3 -299255.559}
SPL {X  -159.990, Y  +527.746, Z    +0.000, E1  +407.012, E3 -299264.832}
SPL {X  -159.990, Y  +533.771, Z    +0.000, E1  +407.034, E3 -299276.717}
SPL {X  -159.990, Y  +542.379, Z    +0.000, E1  +407.067, E3 -299293.687}
SPL {X  -159.990, Y  +549.846, Z    +0.000, E1  +407.016, E3 -299308.532}
SPL {X  -159.990, Y  +554.843, Z    +0.000, E1  +407.014, E3 -299318.410}
SPL {X  -159.990, Y  +560.453, Z    +0.000, E1  +407.023, E3 -299329.493}
SPL {X  -159.990, Y  +566.612, Z    +0.000, E1  +407.022, E3 -299341.675}
SPL {X  -159.990, Y  +572.901, Z    +0.000, E1  +407.028, E3 -299354.087}
SPL {X  -159.990, Y  +578.640, Z    +0.000, E1  +407.021, E3 -299365.439}
SPL {X  -159.990, Y  +583.515, Z    +0.000, E1  +407.019, E3 -299375.078}
SPL {X  -159.990, Y  +589.675, Z    +0.000, E1  +407.042, E3 -299387.216}
SPL {X  -159.990, Y  +596.627, Z    +0.000, E1  +407.034, E3 -299400.956}
SPL {X  -159.990, Y  +602.039, Z    +0.000, E1  +407.021, E3 -299411.663}
SPL {X  -159.990, Y  +607.106, Z    +0.000, E1  +407.028, E3 -299421.670}
SPL {X  -159.990, Y  +612.418, Z    +0.000, E1  +407.023, E3 -299432.182}
SPL {X  -159.990, Y  +618.496, Z    +0.000, E1  +407.049, E3 -299444.148}
SPL {X  -159.990, Y  +624.357, Z    +0.000, E1  +407.020, E3 -299455.774}
SPL {X  -159.990, Y  +629.711, Z    +0.000, E1  +407.034, E3 -299466.343}
SPL {X  -159.990, Y  +635.041, Z    +0.000, E1  +407.022, E3 -299476.888}
SPL {X  -159.990, Y  +639.998, Z    +0.000, E1  +407.027, E3 -299486.680}
SPL {X  -159.990, Y  +646.188, Z    +0.000, E1  +407.041, E3 -299498.906}
SPL {X  -159.990, Y  +652.067, Z    +0.000, E1  +407.023, E3 -299510.542}
SPL {X  -159.990, Y  +657.109, Z    +0.000, E1  +407.025, E3 -299520.521}
SPL {X  -159.990, Y  +662.651, Z    +0.000, E1  +407.027, E3 -299531.477}
SPL {X  -159.990, Y  +668.015, Z    +0.000, E1  +407.025, E3 -299542.077}
SPL {X  -159.972, Y  +673.909, Z    +0.000, E1  +407.029, E3 -299553.742}
SPL {X  -159.776, Y  +679.772, Z    +0.000, E1  +406.992, E3 -299565.543}
SPL {X  -159.384, Y  +685.411, Z    +0.000, E1  +406.921, E3 -299577.105}
SPL {X  -158.642, Y  +692.228, Z    +0.000, E1  +406.819, E3 -299591.320}
SPL {X  -157.651, Y  +698.760, Z    +0.000, E1  +406.609, E3 -299605.315}
SPL {X  -156.719, Y  +703.686, Z    +0.000, E1  +406.438, E3 -299616.008}
SPL {X  -155.778, Y  +707.970, Z    +0.000, E1  +406.262, E3 -299625.483}
SPL {X  -154.419, Y  +713.351, Z    +0.000, E1  +406.025, E3 -299637.514}
SPL {X  -152.913, Y  +718.557, Z    +0.000, E1  +405.729, E3 -299649.366}
SPL {X  -151.262, Y  +723.621, Z    +0.000, E1  +405.429, E3 -299661.032}
SPL {X  -149.074, Y  +729.584, Z    +0.000, E1  +405.040, E3 -299674.961}
SPL {X  -142.577, Y  +744.086, Z    +0.000, E1  +400.686, E3 -299741.167}
ENDSPLINE

SPLINE
SPL {X  -152.566, Y  +719.671, Z    +0.000, E1  +387.682, E3 -299811.638}
SPL {X  -158.253, Y  +695.011, Z    +0.000, E1  +375.913, E3 -299828.310}
SPL {X  -159.486, Y  +684.192, Z    +0.000, E1  +369.965, E3 -299832.256}
SPL {X  -159.898, Y  +676.924, Z    +0.000, E1  +365.683, E3 -299833.954}
SPL {X  -159.990, Y  +671.720, Z    +0.000, E1  +362.298, E3 -299834.794}
SPL {X  -159.990, Y  +668.164, Z    +0.000, E1  +359.695, E3 -299835.210}
SPL {X  -159.990, Y  +665.062, Z    +0.000, E1  +356.961, E3 -299835.549}
SPL {X  -159.990, Y  +660.795, Z    +0.000, E1  +352.651, E3 -299836.212}
SPL {X  -159.990, Y  +654.574, Z    +0.000, E1  +345.673, E3 -299837.667}
SPL {X  -159.990, Y  +647.816, Z    +0.000, E1  +338.252, E3 -299839.918}
SPL {X  -159.990, Y  +640.751, Z    +0.000, E1  +331.747, E3 -299843.512}
SPL {X  -159.990, Y  +611.706, Z    +0.000, E1  +317.244, E3 -299866.285}
SPL {X  -159.990, Y  +567.814, Z    +0.000, E1  +312.360, E3 -299926.375}
SPL {X  -159.990, Y  +558.774, Z    +0.000, E1  +312.384, E3 -299943.941}
SPL {X  -159.990, Y  +550.551, Z    +0.000, E1  +312.385, E3 -299959.882}
SPL {X  -159.990, Y  +542.502, Z    +0.000, E1  +312.392, E3 -299975.497}
SPL {X  -159.990, Y  +536.986, Z    +0.000, E1  +312.423, E3 -299986.217}
SPL {X  -159.990, Y  +532.938, Z    +0.000, E1  +312.415, E3 -299994.043}
SPL {X  -159.990, Y  +525.893, Z    +0.000, E1  +312.375, E3 -300007.657}
SPL {X  -159.990, Y  +518.864, Z    +0.000, E1  +312.415, E3 -300021.339}
SPL {X  -159.990, Y  +512.328, Z    +0.000, E1  +312.388, E3 -300033.973}
SPL {X  -159.990, Y  +505.755, Z    +0.000, E1  +312.413, E3 -300046.750}
ENDSPLINE

SPLINE
SPL {X  -159.990, Y  +517.758, Z    +0.000, E1  +318.109, E3 -300054.473}
ENDSPLINE

SPLINE
SPL {X  -159.990, Y  +516.975, Z    +0.000, E1  +319.588, E3 -300065.537}
SPL {X  -159.990, Y  +508.583, Z    +0.000, E1  +318.552, E3 -300079.842}
SPL {X  -159.990, Y  +499.983, Z    +0.000, E1  +317.561, E3 -300094.296}
SPL {X  -159.990, Y  +492.624, Z    +0.000, E1  +316.776, E3 -300106.400}
SPL {X  -159.990, Y  +485.551, Z    +0.000, E1  +316.053, E3 -300117.949}
SPL {X  -159.990, Y  +477.585, Z    +0.000, E1  +315.156, E3 -300129.860}
SPL {X  -159.990, Y  +470.785, Z    +0.000, E1  +314.453, E3 -300140.033}
SPL {X  -159.990, Y  +463.371, Z    +0.000, E1  +313.690, E3 -300150.758}
SPL {X  -159.990, Y  +455.469, Z    +0.000, E1  +312.807, E3 -300161.284}
SPL {X  -159.990, Y  +445.848, Z    +0.000, E1  +311.866, E3 -300174.376}
SPL {X  -159.990, Y  +436.400, Z    +0.000, E1  +311.449, E3 -300189.758}
SPL {X  -159.990, Y  +429.614, Z    +0.000, E1  +311.486, E3 -300202.548}
SPL {X  -159.990, Y  +423.677, Z    +0.000, E1  +311.471, E3 -300213.660}
SPL {X  -159.990, Y  +417.714, Z    +0.000, E1  +311.484, E3 -300224.870}
SPL {X  -159.990, Y  +412.449, Z    +0.000, E1  +311.483, E3 -300234.730}
SPL {X  -159.990, Y  +406.256, Z    +0.000, E1  +311.459, E3 -300246.298}
SPL {X  -159.990, Y  +399.971, Z    +0.000, E1  +311.480, E3 -300258.113}
SPL {X  -159.990, Y  +394.711, Z    +0.000, E1  +311.476, E3 -300267.971}
SPL {X  -159.990, Y  +387.710, Z    +0.000, E1  +311.455, E3 -300281.094}
SPL {X  -159.966, Y  +379.751, Z    +0.000, E1  +311.465, E3 -300296.058}
SPL {X  -159.734, Y  +373.449, Z    +0.000, E1  +311.528, E3 -300308.162}
SPL {X  -159.230, Y  +366.920, Z    +0.000, E1  +311.592, E3 -300320.905}
SPL {X  -158.532, Y  +360.951, Z    +0.000, E1  +311.745, E3 -300332.879}
SPL {X  -157.692, Y  +355.479, Z    +0.000, E1  +311.882, E3 -300344.007}
SPL {X  -156.349, Y  +348.560, Z    +0.000, E1  +312.101, E3 -300358.346}
SPL {X  -154.984, Y  +342.790, Z    +0.000, E1  +312.392, E3 -300370.643}
SPL {X  -153.247, Y  +336.540, Z    +0.000, E1  +312.660, E3 -300384.079}
SPL {X  -150.765, Y  +328.959, Z    +0.000, E1  +313.136, E3 -300400.825}
SPL {X  -148.834, Y  +323.804, Z    +0.000, E1  +313.556, E3 -300412.478}
SPL {X  -147.343, Y  +320.157, Z    +0.000, E1  +313.838, E3 -300420.768}
SPL {X  -142.380, Y  +309.529, Z    +0.000, E1  +319.953, E3 -300493.528}
ENDSPLINE

SPLINE
SPL {X  -153.420, Y  +337.122, Z    +0.000, E1  +333.501, E3 -300551.026}
SPL {X  -157.288, Y  +353.220, Z    +0.000, E1  +341.134, E3 -300563.071}
SPL {X  -159.049, Y  +365.172, Z    +0.000, E1  +347.392, E3 -300568.625}
SPL {X  -159.749, Y  +373.719, Z    +0.000, E1  +352.250, E3 -300571.245}
SPL {X  -159.988, Y  +381.741, Z    +0.000, E1  +357.172, E3 -300572.720}
SPL {X  -159.990, Y  +387.352, Z    +0.000, E1  +361.387, E3 -300573.422}
SPL {X  -159.990, Y  +391.188, Z    +0.000, E1  +365.082, E3 -300573.963}
SPL {X  -159.990, Y  +395.106, Z    +0.000, E1  +369.154, E3 -300574.704}
SPL {X  -159.990, Y  +400.303, Z    +0.000, E1  +374.927, E3 -300576.025}
SPL {X  -159.990, Y  +408.423, Z    +0.000, E1  +383.302, E3 -300579.104}
SPL {X  -159.990, Y  +438.418, Z    +0.000, E1  +401.067, E3 -300600.677}
SPL {X  -159.990, Y  +482.913, Z    +0.000, E1  +407.036, E3 -300660.031}
SPL {X  -159.990, Y  +489.230, Z    +0.000, E1  +407.019, E3 -300672.543}
SPL {X  -159.990, Y  +495.241, Z    +0.000, E1  +407.026, E3 -300684.422}
SPL {X  -159.990, Y  +501.001, Z    +0.000, E1  +407.020, E3 -300695.799}
SPL {X  -159.990, Y  +506.758, Z    +0.000, E1  +407.038, E3 -300707.145}
SPL {X  -159.990, Y  +512.807, Z    +0.000, E1  +407.022, E3 -300719.136}
SPL {X  -159.990, Y  +518.043, Z    +0.000, E1  +407.016, E3 -300729.514}
SPL {X  -159.990, Y  +523.058, Z    +0.000, E1  +407.015, E3 -300739.430}
SPL {X  -159.990, Y  +527.746, Z    +0.000, E1  +407.012, E3 -300748.703}
SPL {X  -159.990, Y  +533.771, Z    +0.000, E1  +407.034, E3 -300760.588}
SPL {X  -159.990, Y  +542.379, Z    +0.000, E1  +407.067, E3 -300777.557}
SPL {X  -159.990, Y  +549.846, Z    +0.000, E1  +407.016, E3 -300792.403}
SPL {X  -159.990, Y  +554.843, Z    +0.000, E1  +407.014, E3 -300802.281}
SPL {X  -159.990, Y  +560.453, Z    +0.000, E1  +407.023, E3 -300813.364}
SPL {X  -159.990, Y  +566.612, Z    +0.000, E1  +407.022, E3 -300825.546}
SPL {X  -159.990, Y  +572.901, Z    +0.000, E1  +407.028, E3 -300837.958}
SPL {X  -159.990, Y  +578.640, Z    +0.000, E1  +407.021, E3 -300849.310}
SPL {X  -159.990, Y  +583.515, Z    +0.000, E1  +407.019, E3 -300858.949}
SPL {X  -159.990, Y  +589.675, Z    +0.000, E1  +407.042, E3 -300871.087}
SPL {X  -159.990, Y  +596.627, Z    +0.000, E1  +407.034, E3 -300884.827}
SPL {X  -159.990, Y  +602.039, Z    +0.000, E1  +407.021, E3 -300895.534}
SPL {X  -159.990, Y  +607.106, Z    +0.000, E1  +407.028, E3 -300905.541}
SPL {X  -159.990, Y  +612.418, Z    +0.000, E1  +407.023, E3 -300916.053}
SPL {X  -159.990, Y  +618.496, Z    +0.000, E1  +407.049, E3 -300928.019}
SPL {X  -159.990, Y  +624.357, Z    +0.000, E1  +407.020, E3 -300939.645}
SPL {X  -159.990, Y  +629.711, Z    +0.000, E1  +407.034, E3 -300950.214}
SPL {X  -159.990, Y  +635.041, Z    +0.000, E1  +407.022, E3 -300960.759}
SPL {X  -159.990, Y  +639.998, Z    +0.000, E1  +407.027, E3 -300970.551}
SPL {X  -159.990, Y  +646.188, Z    +0.000, E1  +407.041, E3 -300982.777}
SPL {X  -159.990, Y  +652.067, Z    +0.000, E1  +407.023, E3 -300994.413}
SPL {X  -159.990, Y  +657.109, Z    +0.000, E1  +407.025, E3 -301004.392}
SPL {X  -159.990, Y  +662.651, Z    +0.000, E1  +407.027, E3 -301015.348}
SPL {X  -159.990, Y  +668.015, Z    +0.000, E1  +407.025, E3 -301025.948}
SPL {X  -159.972, Y  +673.909, Z    +0.000, E1  +407.029, E3 -301037.613}
SPL {X  -159.776, Y  +679.772, Z    +0.000, E1  +406.992, E3 -301049.414}
SPL {X  -159.384, Y  +685.411, Z    +0.000, E1  +406.921, E3 -301060.976}
SPL {X  -158.839, Y  +690.657, Z    +0.000, E1  +406.819, E3 -301071.930}
SPL {X  -157.875, Y  +697.431, Z    +0.000, E1  +406.688, E3 -301086.270}
SPL {X  -156.719, Y  +703.686, Z    +0.000, E1  +406.438, E3 -301099.879}
SPL {X  -155.778, Y  +707.970, Z    +0.000, E1  +406.262, E3 -301109.353}
SPL {X  -154.419, Y  +713.351, Z    +0.000, E1  +406.025, E3 -301121.385}
SPL {X  -152.913, Y  +718.557, Z    +0.000, E1  +405.729, E3 -301133.237}
SPL {X  -151.262, Y  +723.621, Z    +0.000, E1  +405.429, E3 -301144.903}
SPL {X  -149.074, Y  +729.584, Z    +0.000, E1  +405.040, E3 -301158.832}
SPL {X  -142.577, Y  +744.086, Z    +0.000, E1  +400.686, E3 -301225.038}
ENDSPLINE

SPLINE
SPL {X  -152.566, Y  +719.671, Z    +0.000, E1  +387.682, E3 -301295.509}
SPL {X  -158.253, Y  +695.011, Z    +0.000, E1  +375.913, E3 -301312.181}
SPL {X  -159.486, Y  +684.192, Z    +0.000, E1  +369.965, E3 -301316.127}
SPL {X  -159.898, Y  +676.924, Z    +0.000, E1  +365.683, E3 -301317.825}
SPL {X  -159.990, Y  +671.720, Z    +0.000, E1  +362.298, E3 -301318.665}
SPL {X  -159.990, Y  +668.164, Z    +0.000, E1  +359.695, E3 -301319.081}
SPL {X  -159.990, Y  +665.062, Z    +0.000, E1  +356.961, E3 -301319.420}
SPL {X  -159.990, Y  +660.795, Z    +0.000, E1  +352.651, E3 -301320.083}
SPL {X  -159.990, Y  +654.574, Z    +0.000, E1  +345.673, E3 -301321.538}
SPL {X  -159.990, Y  +647.816, Z    +0.000, E1  +338.252, E3 -301323.789}
SPL {X  -159.990, Y  +640.751, Z    +0.000, E1  +331.747, E3 -301327.383}
SPL {X  -159.990, Y  +611.706, Z    +0.000, E1  +317.244, E3 -301350.156}
SPL {X  -159.990, Y  +567.814, Z    +0.000, E1  +312.360, E3 -301410.246}
SPL {X  -159.990, Y  +558.774, Z    +0.000, E1  +312.384, E3 -301427.812}
SPL {X  -159.990, Y  +550.551, Z    +0.000, E1  +312.385, E3 -301443.753}
SPL {X  -159.990, Y  +542.502, Z    +0.000, E1  +312.392, E3 -301459.367}
SPL {X  -159.990, Y  +536.986, Z    +0.000, E1  +312.423, E3 -301470.088}
SPL {X  -159.990, Y  +532.938, Z    +0.000, E1  +312.415, E3 -301477.914}
SPL {X  -159.990, Y  +525.893, Z    +0.000, E1  +312.375, E3 -301491.528}
SPL {X  -159.990, Y  +518.864, Z    +0.000, E1  +312.415, E3 -301505.210}
SPL {X  -159.990, Y  +512.328, Z    +0.000, E1  +312.388, E3 -301517.844}
SPL {X  -159.990, Y  +505.755, Z    +0.000, E1  +312.413, E3 -301530.621}
ENDSPLINE

SPLINE
SPL {X  -159.990, Y  +517.758, Z    +0.000, E1  +318.109, E3 -301538.344}
ENDSPLINE

SPLINE
SPL {X  -159.990, Y  +516.975, Z    +0.000, E1  +319.588, E3 -301549.408}
SPL {X  -159.990, Y  +508.583, Z    +0.000, E1  +318.552, E3 -301563.713}
SPL {X  -159.990, Y  +499.983, Z    +0.000, E1  +317.561, E3 -301578.167}
SPL {X  -159.990, Y  +492.624, Z    +0.000, E1  +316.776, E3 -301590.271}
SPL {X  -159.990, Y  +485.551, Z    +0.000, E1  +316.053, E3 -301601.820}
SPL {X  -159.990, Y  +477.585, Z    +0.000, E1  +315.156, E3 -301613.731}
SPL {X  -159.990, Y  +470.785, Z    +0.000, E1  +314.453, E3 -301623.904}
SPL {X  -159.990, Y  +463.371, Z    +0.000, E1  +313.690, E3 -301634.629}
SPL {X  -159.990, Y  +455.469, Z    +0.000, E1  +312.807, E3 -301645.155}
SPL {X  -159.990, Y  +445.848, Z    +0.000, E1  +311.866, E3 -301658.247}
SPL {X  -159.990, Y  +436.400, Z    +0.000, E1  +311.449, E3 -301673.629}
SPL {X  -159.990, Y  +429.614, Z    +0.000, E1  +311.486, E3 -301686.419}
SPL {X  -159.990, Y  +423.677, Z    +0.000, E1  +311.471, E3 -301697.531}
SPL {X  -159.990, Y  +417.714, Z    +0.000, E1  +311.484, E3 -301708.741}
SPL {X  -159.990, Y  +412.449, Z    +0.000, E1  +311.483, E3 -301718.601}
SPL {X  -159.990, Y  +406.256, Z    +0.000, E1  +311.459, E3 -301730.169}
SPL {X  -159.990, Y  +399.971, Z    +0.000, E1  +311.480, E3 -301741.984}
SPL {X  -159.990, Y  +394.711, Z    +0.000, E1  +311.476, E3 -301751.842}
SPL {X  -159.990, Y  +387.710, Z    +0.000, E1  +311.455, E3 -301764.965}
SPL {X  -159.966, Y  +379.751, Z    +0.000, E1  +311.465, E3 -301779.929}
SPL {X  -159.734, Y  +373.449, Z    +0.000, E1  +311.528, E3 -301792.033}
SPL {X  -159.230, Y  +366.920, Z    +0.000, E1  +311.592, E3 -301804.776}
SPL {X  -158.532, Y  +360.951, Z    +0.000, E1  +311.745, E3 -301816.750}
SPL {X  -157.692, Y  +355.479, Z    +0.000, E1  +311.882, E3 -301827.878}
SPL {X  -156.349, Y  +348.560, Z    +0.000, E1  +312.101, E3 -301842.217}
SPL {X  -154.984, Y  +342.790, Z    +0.000, E1  +312.392, E3 -301854.514}
SPL {X  -153.247, Y  +336.540, Z    +0.000, E1  +312.660, E3 -301867.950}
SPL {X  -150.765, Y  +328.959, Z    +0.000, E1  +313.136, E3 -301884.696}
SPL {X  -148.834, Y  +323.804, Z    +0.000, E1  +313.556, E3 -301896.349}
SPL {X  -147.343, Y  +320.157, Z    +0.000, E1  +313.838, E3 -301904.638}
SPL {X  -142.380, Y  +309.529, Z    +0.000, E1  +319.953, E3 -301977.399}
ENDSPLINE

SPLINE
SPL {X  -153.420, Y  +337.122, Z    +0.000, E1  +333.501, E3 -302034.897}
SPL {X  -157.288, Y  +353.220, Z    +0.000, E1  +341.134, E3 -302046.942}
SPL {X  -159.049, Y  +365.172, Z    +0.000, E1  +347.392, E3 -302052.496}
SPL {X  -159.749, Y  +373.719, Z    +0.000, E1  +352.250, E3 -302055.116}
SPL {X  -159.988, Y  +381.741, Z    +0.000, E1  +357.172, E3 -302056.591}
SPL {X  -159.990, Y  +387.352, Z    +0.000, E1  +361.387, E3 -302057.293}
SPL {X  -159.990, Y  +391.188, Z    +0.000, E1  +365.082, E3 -302057.834}
SPL {X  -159.990, Y  +395.106, Z    +0.000, E1  +369.154, E3 -302058.575}
SPL {X  -159.990, Y  +400.303, Z    +0.000, E1  +374.927, E3 -302059.896}
SPL {X  -159.990, Y  +408.423, Z    +0.000, E1  +383.302, E3 -302062.975}
SPL {X  -159.990, Y  +438.418, Z    +0.000, E1  +401.067, E3 -302084.548}
SPL {X  -159.990, Y  +482.913, Z    +0.000, E1  +407.036, E3 -302143.902}
SPL {X  -159.990, Y  +489.230, Z    +0.000, E1  +407.019, E3 -302156.414}
SPL {X  -159.990, Y  +495.241, Z    +0.000, E1  +407.026, E3 -302168.293}
SPL {X  -159.990, Y  +501.001, Z    +0.000, E1  +407.020, E3 -302179.670}
SPL {X  -159.990, Y  +506.758, Z    +0.000, E1  +407.038, E3 -302191.016}
SPL {X  -159.990, Y  +512.807, Z    +0.000, E1  +407.022, E3 -302203.007}
SPL {X  -159.990, Y  +518.043, Z    +0.000, E1  +407.016, E3 -302213.385}
SPL {X  -159.990, Y  +523.058, Z    +0.000, E1  +407.015, E3 -302223.301}
SPL {X  -159.990, Y  +527.746, Z    +0.000, E1  +407.012, E3 -302232.574}
SPL {X  -159.990, Y  +533.771, Z    +0.000, E1  +407.034, E3 -302244.459}
SPL {X  -159.990, Y  +542.379, Z    +0.000, E1  +407.067, E3 -302261.428}
SPL {X  -159.990, Y  +549.846, Z    +0.000, E1  +407.016, E3 -302276.274}
SPL {X  -159.990, Y  +554.843, Z    +0.000, E1  +407.014, E3 -302286.152}
SPL {X  -159.990, Y  +560.453, Z    +0.000, E1  +407.023, E3 -302297.235}
SPL {X  -159.990, Y  +566.612, Z    +0.000, E1  +407.022, E3 -302309.417}
SPL {X  -159.990, Y  +572.901, Z    +0.000, E1  +407.028, E3 -302321.829}
SPL {X  -159.990, Y  +578.640, Z    +0.000, E1  +407.021, E3 -302333.180}
SPL {X  -159.990, Y  +583.515, Z    +0.000, E1  +407.019, E3 -302342.820}
SPL {X  -159.990, Y  +589.675, Z    +0.000, E1  +407.042, E3 -302354.958}
SPL {X  -159.990, Y  +596.627, Z    +0.000, E1  +407.034, E3 -302368.698}
SPL {X  -159.990, Y  +602.039, Z    +0.000, E1  +407.021, E3 -302379.405}
SPL {X  -159.990, Y  +607.106, Z    +0.000, E1  +407.028, E3 -302389.412}
SPL {X  -159.990, Y  +612.418, Z    +0.000, E1  +407.023, E3 -302399.924}
SPL {X  -159.990, Y  +618.496, Z    +0.000, E1  +407.049, E3 -302411.890}
SPL {X  -159.990, Y  +624.357, Z    +0.000, E1  +407.020, E3 -302423.516}
SPL {X  -159.990, Y  +629.711, Z    +0.000, E1  +407.034, E3 -302434.085}
SPL {X  -159.990, Y  +635.041, Z    +0.000, E1  +407.022, E3 -302444.630}
SPL {X  -159.990, Y  +639.998, Z    +0.000, E1  +407.027, E3 -302454.422}
SPL {X  -159.990, Y  +646.188, Z    +0.000, E1  +407.041, E3 -302466.648}
SPL {X  -159.990, Y  +652.067, Z    +0.000, E1  +407.023, E3 -302478.284}
SPL {X  -159.990, Y  +657.109, Z    +0.000, E1  +407.025, E3 -302488.263}
SPL {X  -159.990, Y  +662.651, Z    +0.000, E1  +407.027, E3 -302499.219}
SPL {X  -159.990, Y  +668.015, Z    +0.000, E1  +407.025, E3 -302509.819}
SPL {X  -159.972, Y  +673.909, Z    +0.000, E1  +407.029, E3 -302521.484}
SPL {X  -159.776, Y  +679.772, Z    +0.000, E1  +406.992, E3 -302533.285}
SPL {X  -159.384, Y  +685.411, Z    +0.000, E1  +406.921, E3 -302544.847}
SPL {X  -158.839, Y  +690.657, Z    +0.000, E1  +406.819, E3 -302555.801}
SPL {X  -157.875, Y  +697.431, Z    +0.000, E1  +406.688, E3 -302570.141}
SPL {X  -156.719, Y  +703.686, Z    +0.000, E1  +406.438, E3 -302583.750}
SPL {X  -155.778, Y  +707.970, Z    +0.000, E1  +406.262, E3 -302593.224}
SPL {X  -154.419, Y  +713.351, Z    +0.000, E1  +406.025, E3 -302605.256}
SPL {X  -152.913, Y  +718.557, Z    +0.000, E1  +405.729, E3 -302617.108}
SPL {X  -151.262, Y  +723.621, Z    +0.000, E1  +405.429, E3 -302628.774}
SPL {X  -149.074, Y  +729.584, Z    +0.000, E1  +405.040, E3 -302642.703}
SPL {X  -142.577, Y  +744.086, Z    +0.000, E1  +400.686, E3 -302708.909}
ENDSPLINE

SPLINE
SPL {X  -152.566, Y  +719.671, Z    +0.000, E1  +387.682, E3 -302779.380}
SPL {X  -158.253, Y  +695.011, Z    +0.000, E1  +375.913, E3 -302796.052}
SPL {X  -159.486, Y  +684.192, Z    +0.000, E1  +369.965, E3 -302799.998}
SPL {X  -159.898, Y  +676.924, Z    +0.000, E1  +365.683, E3 -302801.696}
SPL {X  -159.990, Y  +671.720, Z    +0.000, E1  +362.298, E3 -302802.536}
SPL {X  -159.990, Y  +668.164, Z    +0.000, E1  +359.695, E3 -302802.952}
SPL {X  -159.990, Y  +665.062, Z    +0.000, E1  +356.961, E3 -302803.291}
SPL {X  -159.990, Y  +660.795, Z    +0.000, E1  +352.651, E3 -302803.954}
SPL {X  -159.990, Y  +654.574, Z    +0.000, E1  +345.673, E3 -302805.409}
SPL {X  -159.990, Y  +647.816, Z    +0.000, E1  +338.252, E3 -302807.660}
SPL {X  -159.990, Y  +640.751, Z    +0.000, E1  +331.747, E3 -302811.254}
SPL {X  -159.990, Y  +611.706, Z    +0.000, E1  +317.244, E3 -302834.027}
SPL {X  -159.990, Y  +567.814, Z    +0.000, E1  +312.360, E3 -302894.117}
SPL {X  -159.990, Y  +558.774, Z    +0.000, E1  +312.384, E3 -302911.683}
SPL {X  -159.990, Y  +550.551, Z    +0.000, E1  +312.385, E3 -302927.624}
SPL {X  -159.990, Y  +542.502, Z    +0.000, E1  +312.392, E3 -302943.238}
SPL {X  -159.990, Y  +536.986, Z    +0.000, E1  +312.423, E3 -302953.959}
SPL {X  -159.990, Y  +532.938, Z    +0.000, E1  +312.415, E3 -302961.785}
SPL {X  -159.990, Y  +525.893, Z    +0.000, E1  +312.375, E3 -302975.399}
SPL {X  -159.990, Y  +518.864, Z    +0.000, E1  +312.415, E3 -302989.081}
SPL {X  -159.990, Y  +512.328, Z    +0.000, E1  +312.388, E3 -303001.715}
SPL {X  -159.990, Y  +505.755, Z    +0.000, E1  +312.413, E3 -303014.492}
ENDSPLINE

SPLINE
SPL {X  -159.990, Y  +517.758, Z    +0.000, E1  +318.109, E3 -303022.215}
ENDSPLINE

SPLINE
SPL {X  -159.990, Y  +516.975, Z    +0.000, E1  +319.588, E3 -303033.278}
SPL {X  -159.990, Y  +508.583, Z    +0.000, E1  +318.552, E3 -303047.584}
SPL {X  -159.990, Y  +499.983, Z    +0.000, E1  +317.561, E3 -303062.038}
SPL {X  -159.990, Y  +492.624, Z    +0.000, E1  +316.776, E3 -303074.142}
SPL {X  -159.990, Y  +485.551, Z    +0.000, E1  +316.053, E3 -303085.691}
SPL {X  -159.990, Y  +477.585, Z    +0.000, E1  +315.156, E3 -303097.602}
SPL {X  -159.990, Y  +470.785, Z    +0.000, E1  +314.453, E3 -303107.775}
SPL {X  -159.990, Y  +463.371, Z    +0.000, E1  +313.690, E3 -303118.500}
SPL {X  -159.990, Y  +455.469, Z    +0.000, E1  +312.807, E3 -303129.026}
SPL {X  -159.990, Y  +445.848, Z    +0.000, E1  +311.866, E3 -303142.118}
SPL {X  -159.990, Y  +436.400, Z    +0.000, E1  +311.449, E3 -303157.500}
SPL {X  -159.990, Y  +429.614, Z    +0.000, E1  +311.486, E3 -303170.290}
SPL {X  -159.990, Y  +423.677, Z    +0.000, E1  +311.471, E3 -303181.402}
SPL {X  -159.990, Y  +417.714, Z    +0.000, E1  +311.484, E3 -303192.612}
SPL {X  -159.990, Y  +412.449, Z    +0.000, E1  +311.483, E3 -303202.472}
SPL {X  -159.990, Y  +406.256, Z    +0.000, E1  +311.459, E3 -303214.040}
SPL {X  -159.990, Y  +399.971, Z    +0.000, E1  +311.480, E3 -303225.855}
SPL {X  -159.990, Y  +394.711, Z    +0.000, E1  +311.476, E3 -303235.713}
SPL {X  -159.990, Y  +387.710, Z    +0.000, E1  +311.455, E3 -303248.836}
SPL {X  -159.966, Y  +379.751, Z    +0.000, E1  +311.465, E3 -303263.800}
SPL {X  -159.734, Y  +373.449, Z    +0.000, E1  +311.528, E3 -303275.904}
SPL {X  -159.230, Y  +366.920, Z    +0.000, E1  +311.592, E3 -303288.647}
SPL {X  -158.532, Y  +360.951, Z    +0.000, E1  +311.745, E3 -303300.621}
SPL {X  -157.692, Y  +355.479, Z    +0.000, E1  +311.882, E3 -303311.749}
SPL {X  -156.349, Y  +348.560, Z    +0.000, E1  +312.101, E3 -303326.088}
SPL {X  -154.984, Y  +342.790, Z    +0.000, E1  +312.392, E3 -303338.385}
SPL {X  -153.247, Y  +336.540, Z    +0.000, E1  +312.660, E3 -303351.820}
SPL {X  -150.765, Y  +328.959, Z    +0.000, E1  +313.136, E3 -303368.567}
SPL {X  -148.834, Y  +323.804, Z    +0.000, E1  +313.556, E3 -303380.220}
SPL {X  -147.343, Y  +320.157, Z    +0.000, E1  +313.838, E3 -303388.509}
SPL {X  -142.380, Y  +309.529, Z    +0.000, E1  +319.953, E3 -303461.270}
ENDSPLINE

SPLINE
SPL {X  -153.420, Y  +337.122, Z    +0.000, E1  +333.501, E3 -303518.768}
SPL {X  -157.288, Y  +353.220, Z    +0.000, E1  +341.134, E3 -303530.813}
SPL {X  -159.049, Y  +365.172, Z    +0.000, E1  +347.392, E3 -303536.367}
SPL {X  -159.749, Y  +373.719, Z    +0.000, E1  +352.250, E3 -303538.987}
SPL {X  -159.988, Y  +381.741, Z    +0.000, E1  +357.172, E3 -303540.462}
SPL {X  -159.990, Y  +387.352, Z    +0.000, E1  +361.387, E3 -303541.164}
SPL {X  -159.990, Y  +391.188, Z    +0.000, E1  +365.082, E3 -303541.705}
SPL {X  -159.990, Y  +395.106, Z    +0.000, E1  +369.154, E3 -303542.446}
SPL {X  -159.990, Y  +400.303, Z    +0.000, E1  +374.927, E3 -303543.767}
SPL {X  -159.990, Y  +408.423, Z    +0.000, E1  +383.302, E3 -303546.846}
SPL {X  -159.990, Y  +438.418, Z    +0.000, E1  +401.067, E3 -303568.419}
SPL {X  -159.990, Y  +482.913, Z    +0.000, E1  +407.036, E3 -303627.773}
SPL {X  -159.990, Y  +489.230, Z    +0.000, E1  +407.019, E3 -303640.285}
SPL {X  -159.990, Y  +495.241, Z    +0.000, E1  +407.026, E3 -303652.164}
SPL {X  -159.990, Y  +501.001, Z    +0.000, E1  +407.020, E3 -303663.541}
SPL {X  -159.990, Y  +506.758, Z    +0.000, E1  +407.038, E3 -303674.887}
SPL {X  -159.990, Y  +512.807, Z    +0.000, E1  +407.022, E3 -303686.878}
SPL {X  -159.990, Y  +518.043, Z    +0.000, E1  +407.016, E3 -303697.256}
SPL {X  -159.990, Y  +523.058, Z    +0.000, E1  +407.015, E3 -303707.171}
SPL {X  -159.990, Y  +527.746, Z    +0.000, E1  +407.012, E3 -303716.445}
SPL {X  -159.990, Y  +533.771, Z    +0.000, E1  +407.034, E3 -303728.330}
SPL {X  -159.990, Y  +542.379, Z    +0.000, E1  +407.067, E3 -303745.299}
SPL {X  -159.990, Y  +549.846, Z    +0.000, E1  +407.016, E3 -303760.145}
SPL {X  -159.990, Y  +554.843, Z    +0.000, E1  +407.014, E3 -303770.023}
SPL {X  -159.990, Y  +560.453, Z    +0.000, E1  +407.023, E3 -303781.106}
SPL {X  -159.990, Y  +566.612, Z    +0.000, E1  +407.022, E3 -303793.288}
SPL {X  -159.990, Y  +572.901, Z    +0.000, E1  +407.028, E3 -303805.700}
SPL {X  -159.990, Y  +578.640, Z    +0.000, E1  +407.021, E3 -303817.051}
SPL {X  -159.990, Y  +583.515, Z    +0.000, E1  +407.019, E3 -303826.691}
SPL {X  -159.990, Y  +589.675, Z    +0.000, E1  +407.042, E3 -303838.829}
SPL {X  -159.990, Y  +596.627, Z    +0.000, E1  +407.034, E3 -303852.569}
SPL {X  -159.990, Y  +602.039, Z    +0.000, E1  +407.021, E3 -303863.276}
SPL {X  -159.990, Y  +607.106, Z    +0.000, E1  +407.028, E3 -303873.283}
SPL {X  -159.990, Y  +612.418, Z    +0.000, E1  +407.023, E3 -303883.795}
SPL {X  -159.990, Y  +618.496, Z    +0.000, E1  +407.049, E3 -303895.761}
SPL {X  -159.990, Y  +624.357, Z    +0.000, E1  +407.020, E3 -303907.387}
SPL {X  -159.990, Y  +629.711, Z    +0.000, E1  +407.034, E3 -303917.956}
SPL {X  -159.990, Y  +635.041, Z    +0.000, E1  +407.022, E3 -303928.501}
SPL {X  -159.990, Y  +639.998, Z    +0.000, E1  +407.027, E3 -303938.293}
SPL {X  -159.990, Y  +646.188, Z    +0.000, E1  +407.041, E3 -303950.519}
SPL {X  -159.990, Y  +652.067, Z    +0.000, E1  +407.023, E3 -303962.155}
SPL {X  -159.990, Y  +657.109, Z    +0.000, E1  +407.025, E3 -303972.134}
SPL {X  -159.990, Y  +662.651, Z    +0.000, E1  +407.027, E3 -303983.090}
SPL {X  -159.990, Y  +668.015, Z    +0.000, E1  +407.025, E3 -303993.690}
SPL {X  -159.972, Y  +673.909, Z    +0.000, E1  +407.029, E3 -304005.355}
SPL {X  -159.776, Y  +679.772, Z    +0.000, E1  +406.992, E3 -304017.156}
SPL {X  -159.384, Y  +685.411, Z    +0.000, E1  +406.921, E3 -304028.718}
SPL {X  -158.839, Y  +690.657, Z    +0.000, E1  +406.819, E3 -304039.672}
SPL {X  -157.875, Y  +697.431, Z    +0.000, E1  +406.688, E3 -304054.011}
SPL {X  -156.719, Y  +703.686, Z    +0.000, E1  +406.438, E3 -304067.621}
SPL {X  -155.778, Y  +707.970, Z    +0.000, E1  +406.262, E3 -304077.095}
SPL {X  -154.419, Y  +713.351, Z    +0.000, E1  +406.025, E3 -304089.127}
SPL {X  -152.913, Y  +718.557, Z    +0.000, E1  +405.729, E3 -304100.979}
SPL {X  -151.262, Y  +723.621, Z    +0.000, E1  +405.429, E3 -304112.645}
SPL {X  -149.074, Y  +729.584, Z    +0.000, E1  +405.040, E3 -304126.574}
SPL {X  -142.577, Y  +744.086, Z    +0.000, E1  +400.686, E3 -304192.780}
ENDSPLINE

SPLINE
SPL {X  -152.566, Y  +719.671, Z    +0.000, E1  +387.682, E3 -304263.251}
SPL {X  -158.253, Y  +695.011, Z    +0.000, E1  +375.913, E3 -304279.923}
SPL {X  -159.486, Y  +684.192, Z    +0.000, E1  +369.965, E3 -304283.869}
SPL {X  -159.898, Y  +676.924, Z    +0.000, E1  +365.683, E3 -304285.567}
SPL {X  -159.990, Y  +671.720, Z    +0.000, E1  +362.298, E3 -304286.407}
SPL {X  -159.990, Y  +668.164, Z    +0.000, E1  +359.695, E3 -304286.822}
SPL {X  -159.990, Y  +665.062, Z    +0.000, E1  +356.961, E3 -304287.162}
SPL {X  -159.990, Y  +660.795, Z    +0.000, E1  +352.651, E3 -304287.825}
SPL {X  -159.990, Y  +654.574, Z    +0.000, E1  +345.673, E3 -304289.280}
SPL {X  -159.990, Y  +647.816, Z    +0.000, E1  +338.252, E3 -304291.531}
SPL {X  -159.990, Y  +640.751, Z    +0.000, E1  +331.747, E3 -304295.125}
SPL {X  -159.990, Y  +611.706, Z    +0.000, E1  +317.244, E3 -304317.898}
SPL {X  -159.990, Y  +567.814, Z    +0.000, E1  +312.360, E3 -304377.988}
SPL {X  -159.990, Y  +558.774, Z    +0.000, E1  +312.384, E3 -304395.554}
SPL {X  -159.990, Y  +550.551, Z    +0.000, E1  +312.385, E3 -304411.495}
SPL {X  -159.990, Y  +542.502, Z    +0.000, E1  +312.392, E3 -304427.109}
SPL {X  -159.990, Y  +536.986, Z    +0.000, E1  +312.423, E3 -304437.830}
SPL {X  -159.990, Y  +532.938, Z    +0.000, E1  +312.415, E3 -304445.656}
SPL {X  -159.990, Y  +525.893, Z    +0.000, E1  +312.375, E3 -304459.270}
SPL {X  -159.990, Y  +518.864, Z    +0.000, E1  +312.415, E3 -304472.952}
SPL {X  -159.990, Y  +512.328, Z    +0.000, E1  +312.388, E3 -304485.586}
SPL {X  -159.990, Y  +505.755, Z    +0.000, E1  +312.413, E3 -304498.363}
ENDSPLINE

SPLINE
SPL {X  -159.990, Y  +517.758, Z    +0.000, E1  +318.109, E3 -304506.086}
ENDSPLINE

SPLINE
SPL {X  -159.990, Y  +516.975, Z    +0.000, E1  +319.588, E3 -304517.149}
SPL {X  -159.990, Y  +508.583, Z    +0.000, E1  +318.552, E3 -304531.455}
SPL {X  -159.990, Y  +499.983, Z    +0.000, E1  +317.561, E3 -304545.909}
SPL {X  -159.990, Y  +492.624, Z    +0.000, E1  +316.776, E3 -304558.013}
SPL {X  -159.990, Y  +485.551, Z    +0.000, E1  +316.053, E3 -304569.562}
SPL {X  -159.990, Y  +477.585, Z    +0.000, E1  +315.156, E3 -304581.473}
SPL {X  -159.990, Y  +470.785, Z    +0.000, E1  +314.453, E3 -304591.646}
SPL {X  -159.990, Y  +463.371, Z    +0.000, E1  +313.690, E3 -304602.371}
SPL {X  -159.990, Y  +455.469, Z    +0.000, E1  +312.807, E3 -304612.897}
SPL {X  -159.990, Y  +445.848, Z    +0.000, E1  +311.866, E3 -304625.989}
SPL {X  -159.990, Y  +436.400, Z    +0.000, E1  +311.449, E3 -304641.371}
SPL {X  -159.990, Y  +429.614, Z    +0.000, E1  +311.486, E3 -304654.161}
SPL {X  -159.990, Y  +423.677, Z    +0.000, E1  +311.471, E3 -304665.273}
SPL {X  -159.990, Y  +417.714, Z    +0.000, E1  +311.484, E3 -304676.483}
SPL {X  -159.990, Y  +412.449, Z    +0.000, E1  +311.483, E3 -304686.343}
SPL {X  -159.990, Y  +406.256, Z    +0.000, E1  +311.459, E3 -304697.911}
SPL {X  -159.990, Y  +399.971, Z    +0.000, E1  +311.480, E3 -304709.726}
SPL {X  -159.990, Y  +394.711, Z    +0.000, E1  +311.476, E3 -304719.584}
SPL {X  -159.990, Y  +387.710, Z    +0.000, E1  +311.455, E3 -304732.707}
SPL {X  -159.966, Y  +379.751, Z    +0.000, E1  +311.465, E3 -304747.671}
SPL {X  -159.734, Y  +373.449, Z    +0.000, E1  +311.528, E3 -304759.775}
SPL {X  -159.230, Y  +366.920, Z    +0.000, E1  +311.592, E3 -304772.518}
SPL {X  -158.532, Y  +360.951, Z    +0.000, E1  +311.745, E3 -304784.492}
SPL {X  -157.692, Y  +355.479, Z    +0.000, E1  +311.882, E3 -304795.620}
SPL {X  -156.349, Y  +348.560, Z    +0.000, E1  +312.101, E3 -304809.959}
SPL {X  -154.984, Y  +342.790, Z    +0.000, E1  +312.392, E3 -304822.256}
SPL {X  -153.247, Y  +336.540, Z    +0.000, E1  +312.660, E3 -304835.691}
SPL {X  -150.765, Y  +328.959, Z    +0.000, E1  +313.136, E3 -304852.438}
SPL {X  -148.834, Y  +323.804, Z    +0.000, E1  +313.556, E3 -304864.091}
SPL {X  -147.343, Y  +320.157, Z    +0.000, E1  +313.838, E3 -304872.380}
SPL {X  -142.380, Y  +309.529, Z    +0.000, E1  +319.953, E3 -304945.141}
ENDSPLINE

